	{attribute 'TcIecLibraryType'}
	{attribute 'external_name' := 'F_VN_CalibrateLinescanCameraExp_GUID_4214EBFD_93AA_4917_F265_40A1261014F9'}
	(* Compute the camera parameters (intrinsic + extrinsic) by evaluating images containing a line calibration pattern. The pattern must consist of alternating vertical and diagonal lines, with each diagonal having the same constant slope: |\|\|...\|. The results are only valid for the x-direction of a line scan image. To get accurate x-values for a transformation into world coordinates, the y-coordinate must be set to half the sensor width and so equal to the cy-value of the camera matrix. For other y-values, the results are approximated and can be inaccurate. The extrinsic parameters are computed for the first image in the array. (expert function) *)
	FUNCTION F_VN_CalibrateLinescanCameraExp : HRESULT
	VAR_INPUT
		pSrcImages	:	PVOID;	(* Pointer to an array of 1 or more source images (1 channel). If the images have more than 1 row, each row must contain an image of the same pattern position. *)
		nSrcArraySize	:	UINT;	(* pSrcImages array size *)
		ipPatternLineOrigins	:	ITcVnContainer;	(* X position of the pattern line origins (ContainerType_Vector_REAL, usually same origin for vertical and following diagonal line) *)
		fSlopeRad	:	LREAL;	(* Slope of the diagonal line in rad (> 0, < PI/2), relative to the vertical line (i.e., 0 would be a vertical line, PI/2 a horizontal line) *)
	END_VAR
	VAR_IN_OUT
		aCameraMatrix	:	TcVnMatrix3x3_LREAL;	(* Returns the camera matrix *)
		aDistortionCoefficients	:	TcVnArray8_LREAL;	(* Returns the lens distortion coefficients [k1, k2, p1, p2, k3, k4, k5, k6] *)
		aRotationMatrix	:	TcVnMatrix3x3_LREAL;	(* Returns the rotation matrix *)
		aTranslationVector	:	TcVnVector3_LREAL;	(* Returns the translation vector *)
		fReprojError	:	LREAL;	(* Returns the reprojection error *)
		stCalibrationOptions	:	TcVnCameraCalibrationOptions;	(* Calibration options (recommended to set bFixAspectRatio, bFixPrincipalPoint, bZeroTangentDist) *)
	END_VAR
	VAR_INPUT
		eEdgeDirection	:	ETcVnEdgeDirection;	(* Specification of the edge direction to search for *)
		fMinStrength	:	REAL;	(* Specification of the minimum strength (intensity difference) of the edge to search for *)
		nMaxSearchLines	:	UDINT;	(* Maximum number of search lines (equally distributed over the image height, at most 1 searchline per image row) *)
		nMaxThickness	:	UDINT;	(* Specification of the maximum thickness of the edge to search for, which means fMinStrength must be reached within nMaxThickness pixels *)
		nSubpixelsIterations	:	UDINT;	(* Specifies the number of subpixels (for INTERPOLATION, 10 - 20 usually is sufficient) or maximum number of iterations for optimizing the parameters (for APPROX_ERF and APPROX_GAUSSIAN, 50 - 100 usually is sufficient) *)
		fApproxPrecision	:	REAL;	(* Specifies the approximation precision for APPROX_ERF and APPROX_GAUSSIAN (0.001 usually is sufficient, unused for INTERPOLATION) *)
		eAlgorithm	:	ETcVnEdgeDetectionAlgorithm;	(* Selection of the edge detection algorithm *)
		hrPrev	:	HRESULT;	(* HRESULT indicating the result of previous operations (If SUCCEEDED(hrPrev) equals false, no operation is executed.) *)
	END_VAR

END_FUNCTION

// Functions/Geometric and Coordinate Transformations/Calibration/F_VN_CompensateLensDistortion

	{attribute 'TcIecLibraryType'}
	{attribute 'external_name' := 'F_VN_CompensateLensDistortion_GUID_A7E90272_F769_427D_ED4C_EA7B5F41935C'}
	(* Transforms an image to compensate the lens distortion. *)
	FUNCTION F_VN_CompensateLensDistortion : HRESULT
	VAR_INPUT
		ipSrcImage	:	ITcVnImage;	(* Source image *)
		ipDestImage	:	REFERENCE TO ITcVnImage;	(* Destination image (An appropriate destination image will be created if required.) *)
	END_VAR
	VAR_IN_OUT
		aCameraMatrix	:	TcVnMatrix3x3_LREAL;	(* Camera matrix containing the intrinsic parameters *)
		aDistortionCoefficients	:	TcVnArray4_LREAL;	(* Lens distortion coefficients [k1, k2, p1, p2] *)
	END_VAR
	VAR_INPUT
		hrPrev	:	HRESULT;	(* HRESULT indicating the result of previous operations (If SUCCEEDED(hrPrev) equals false, no operation is executed.) *)
	END_VAR

END_FUNCTION

// Functions/Geometric and Coordinate Transformations/Calibration/F_VN_CompensateLensDistortionExp1

	{attribute 'TcIecLibraryType'}
	{attribute 'external_name' := 'F_VN_CompensateLensDistortionExp1_GUID_3D946475_AB4A_4E66_EAD8_FDBE1E19AFDC'}
	(* Transforms an image to compensate the lens distortion. (expert function) *)
	FUNCTION F_VN_CompensateLensDistortionExp1 : HRESULT
	VAR_INPUT
		ipSrcImage	:	ITcVnImage;	(* Source image *)
		ipDestImage	:	REFERENCE TO ITcVnImage;	(* Destination image (An appropriate destination image will be created if required.) *)
	END_VAR
	VAR_IN_OUT
		aCameraMatrix	:	TcVnMatrix3x3_LREAL;	(* Camera matrix containing the intrinsic parameters *)
		aDistortionCoefficients	:	TcVnArray8_LREAL;	(* Lens distortion coefficients [k1, k2, p1, p2, k3, k4, k5, k6] *)
	END_VAR
	VAR_INPUT
		hrPrev	:	HRESULT;	(* HRESULT indicating the result of previous operations (If SUCCEEDED(hrPrev) equals false, no operation is executed.) *)
	END_VAR

END_FUNCTION

// Functions/Geometric and Coordinate Transformations/Calibration/F_VN_CompensateLensDistortionExp2

	{attribute 'TcIecLibraryType'}
	{attribute 'external_name' := 'F_VN_CompensateLensDistortionExp2_GUID_C20F3BF9_EE4F_4E64_CEDC_52B963B053AC'}
	(* Transforms an image to compensate the lens distortion. (expert function) *)
	FUNCTION F_VN_CompensateLensDistortionExp2 : HRESULT
	VAR_INPUT
		ipSrcImage	:	ITcVnImage;	(* Source image *)
		ipDestImage	:	REFERENCE TO ITcVnImage;	(* Destination image (An appropriate destination image will be created if required.) *)
	END_VAR
	VAR_IN_OUT
		aCameraMatrix	:	TcVnMatrix3x3_LREAL;	(* Camera matrix containing the intrinsic parameters *)
		aDistortionCoefficients	:	TcVnArray8_LREAL;	(* Lens distortion coefficients [k1, k2, p1, p2, k3, k4, k5, k6] *)
		aNewCameraMatrix	:	TcVnMatrix3x3_LREAL;	(* Allows additional scaling and shifting of the result image *)
	END_VAR
	VAR_INPUT
		hrPrev	:	HRESULT;	(* HRESULT indicating the result of previous operations (If SUCCEEDED(hrPrev) equals false, no operation is executed.) *)
	END_VAR

END_FUNCTION

// Functions/Geometric and Coordinate Transformations/Calibration/F_VN_CompensateLensDistortionForPoints

	{attribute 'TcIecLibraryType'}
	{attribute 'external_name' := 'F_VN_CompensateLensDistortionForPoints_GUID_1A71B91E_10E3_4E50_D6FD_7DACBEC96CC6'}
	(* Transforms point coordinates to compensate the lens distortion. *)
	FUNCTION F_VN_CompensateLensDistortionForPoints : HRESULT
	VAR_INPUT
		ipSrcPoints	:	ITcVnContainer;	(* Container with source point coordinates (ContainerType_Vector_TcVnPoint2_REAL or ContainerType_Vector_TcVnPoint2_DINT) *)
		ipDestPoints	:	REFERENCE TO ITcVnContainer;	(* Returns a container with the transformed point coordinates (ContainerType_Vector_TcVnPoint2_REAL) *)
	END_VAR
	VAR_IN_OUT
		aCameraMatrix	:	TcVnMatrix3x3_LREAL;	(* Camera matrix containing the intrinsic parameters *)
		aDistortionCoefficients	:	TcVnArray4_LREAL;	(* Lens distortion coefficients [k1, k2, p1, p2] *)
	END_VAR
	VAR_INPUT
		hrPrev	:	HRESULT;	(* HRESULT indicating the result of previous operations (If SUCCEEDED(hrPrev) equals false, no operation is executed.) *)
	END_VAR

END_FUNCTION

// Functions/Geometric and Coordinate Transformations/Calibration/F_VN_CompensateLensDistortionForPointsExp1

	{attribute 'TcIecLibraryType'}
	{attribute 'external_name' := 'F_VN_CompensateLensDistortionForPointsExp1_GUID_7B846EAA_13D4_4E78_E7DF_523567D8C748'}
	(* Transforms point coordinates to compensate the lens distortion. (expert function) *)
	FUNCTION F_VN_CompensateLensDistortionForPointsExp1 : HRESULT
	VAR_INPUT
		ipSrcPoints	:	ITcVnContainer;	(* Container with source point coordinates (ContainerType_Vector_TcVnPoint2_REAL or ContainerType_Vector_TcVnPoint2_DINT) *)
		ipDestPoints	:	REFERENCE TO ITcVnContainer;	(* Returns a container with the transformed point coordinates (ContainerType_Vector_TcVnPoint2_REAL) *)
	END_VAR
	VAR_IN_OUT
		aCameraMatrix	:	TcVnMatrix3x3_LREAL;	(* Camera matrix containing the intrinsic parameters *)
		aDistortionCoefficients	:	TcVnArray8_LREAL;	(* Lens distortion coefficients [k1, k2, p1, p2, k3, k4, k5, k6] *)
	END_VAR
	VAR_INPUT
		hrPrev	:	HRESULT;	(* HRESULT indicating the result of previous operations (If SUCCEEDED(hrPrev) equals false, no operation is executed.) *)
	END_VAR

END_FUNCTION

// Functions/Geometric and Coordinate Transformations/Calibration/F_VN_CompensateLensDistortionForPointsExp2

	{attribute 'TcIecLibraryType'}
	{attribute 'external_name' := 'F_VN_CompensateLensDistortionForPointsExp2_GUID_34553A45_A6A3_444C_C55B_DC9387F7369D'}
	(* Transforms point coordinates to compensate the lens distortion. (expert function) *)
	FUNCTION F_VN_CompensateLensDistortionForPointsExp2 : HRESULT
	VAR_INPUT
		ipSrcPoints	:	ITcVnContainer;	(* Container with source point coordinates (ContainerType_Vector_TcVnPoint2_REAL or ContainerType_Vector_TcVnPoint2_DINT) *)
		ipDestPoints	:	REFERENCE TO ITcVnContainer;	(* Returns a container with the transformed point coordinates (ContainerType_Vector_TcVnPoint2_REAL) *)
	END_VAR
	VAR_IN_OUT
		aCameraMatrix	:	TcVnMatrix3x3_LREAL;	(* Camera matrix containing the intrinsic parameters *)
		aDistortionCoefficients	:	TcVnArray8_LREAL;	(* Lens distortion coefficients [k1, k2, p1, p2, k3, k4, k5, k6] *)
		aNewCameraMatrix	:	TcVnMatrix3x3_LREAL;	(* Allows additional shifting of the result point coordinates *)
	END_VAR
	VAR_INPUT
		hrPrev	:	HRESULT;	(* HRESULT indicating the result of previous operations (If SUCCEEDED(hrPrev) equals false, no operation is executed.) *)
	END_VAR

END_FUNCTION

// Functions/Geometric and Coordinate Transformations/Calibration/F_VN_DetectPatternPoints

	{attribute 'TcIecLibraryType'}
	{attribute 'external_name' := 'F_VN_DetectPatternPoints_GUID_E1BA4EA3_C273_48EA_C92C_C13F9E969AAA'}
	(* Detects calibration pattern points (circles) within the provided image. *)
	FUNCTION F_VN_DetectPatternPoints : HRESULT
	VAR_INPUT
		ipSrcImage	:	ITcVnImage;	(* Source image (USINT, 1 channel) *)
		ipPatternPoints	:	REFERENCE TO ITcVnContainer;	(* Returns the pattern point positions (ContainerType_Vector_TcVnPoint2_REAL; Non-zero interface pointers are reused.) *)
	END_VAR
	VAR_IN_OUT
		stBlobDetectionParams	:	TcVnParamsBlobDetection;	(* Parameters to detect and filter contours. *)
	END_VAR
	VAR_INPUT
		nNumberOfPoints	:	UDINT;	(* Expected number of pattern points *)
		hrPrev	:	HRESULT;	(* HRESULT indicating the result of previous operations (If SUCCEEDED(hrPrev) equals false, no operation is executed.) *)
	END_VAR

END_FUNCTION

// Functions/Geometric and Coordinate Transformations/Calibration/F_VN_DetectPatternPointsExp

	{attribute 'TcIecLibraryType'}
	{attribute 'external_name' := 'F_VN_DetectPatternPointsExp_GUID_0FD53513_A53D_46BB_DEE5_D943CEECBF42'}
	(* Detects calibration pattern points (circles) within the provided image. (expert function) *)
	FUNCTION F_VN_DetectPatternPointsExp : HRESULT
	VAR_INPUT
		ipSrcImage	:	ITcVnImage;	(* Source image (USINT, 1 channel) *)
		ipPatternPoints	:	REFERENCE TO ITcVnContainer;	(* Returns the pattern point positions (ContainerType_Vector_TcVnPoint2_REAL; Non-zero interface pointers are reused.) *)
	END_VAR
	VAR_IN_OUT
		stBlobDetectionParams	:	TcVnParamsBlobDetection;	(* Parameters to detect and filter contours. *)
	END_VAR
	VAR_INPUT
		nNumberOfPoints	:	UDINT;	(* Expected number of pattern points *)
		fSizeDiffThresFactor	:	REAL;	(* Threshold for filtering contours by average size *)
		bSubpixelAccuracy	:	BOOL;	(* If true, the pattern points are detected with subpixel accuracy *)
		eEdgeDirection	:	ETcVnEdgeDirection;	(* Specification of the edge direction to search for (from center to outside circle) *)
		fMinStrength	:	REAL;	(* Specification of the minimum strength (intensity difference) of the edge to search for *)
		nMaxThickness	:	UDINT;	(* Specification of the maximum thickness of the edge to search for, which means fMinStrength must be reached within nMaxThickness pixels *)
		nSubpixelsIterations	:	UDINT;	(* Specifies the number of subpixels (for INTERPOLATION, 10 - 20 usually is sufficient) or maximum number of iterations for optimizing the parameters (for APPROX_ERF and APPROX_GAUSSIAN, 50 - 100 usually is sufficient) *)
		nSearchLines	:	UDINT;	(* Specifies the amount of search lines, which are equally distributed in all directions (must be >= 8 and a multiple of 4) *)
		fApproxPrecision	:	REAL;	(* Specifies the approximation precision for APPROX_ERF and APPROX_GAUSSIAN (0.001 usually is sufficient, unused for INTERPOLATION) *)
		eAlgorithm	:	ETcVnEdgeDetectionAlgorithm;	(* Selection of the edge detection algorithm *)
		hrPrev	:	HRESULT;	(* HRESULT indicating the result of previous operations (If SUCCEEDED(hrPrev) equals false, no operation is executed.) *)
	END_VAR

END_FUNCTION

// Functions/Geometric and Coordinate Transformations/Calibration/F_VN_GenerateCalibrationPatternReferencePoints

	{attribute 'TcIecLibraryType'}
	{attribute 'external_name' := 'F_VN_GenerateCalibrationPatternReferencePoints_GUID_599A364B_79C4_437C_C2A7_ACD3D87798EB'}
	(* Generate reference points for common calibration patterns. *)
	FUNCTION F_VN_GenerateCalibrationPatternReferencePoints : HRESULT
	VAR_INPUT
		ipReferencePoints	:	REFERENCE TO ITcVnContainer;	(* Returns the generated reference points (ContainerType_Vector_TcVnPoint3_REAL) *)
		ePattern	:	ETcVnCalibrationPattern;	(* Calibration pattern type *)
		eOrigin	:	ETcVnCalibrationPatternOrigin;	(* Calibration pattern origin *)
		nWidth	:	UDINT;	(* Pattern width, i.e. number of pattern points in x direction *)
		nHeight	:	UDINT;	(* Pattern height, i.e. number of pattern points in y direction *)
		fDistX	:	REAL;	(* Distance between pattern points in x direction *)
		fDistY	:	REAL;	(* Distance between pattern points in y direction *)
		hrPrev	:	HRESULT;	(* HRESULT indicating the result of previous operations (If SUCCEEDED(hrPrev) equals false, no operation is executed.) *)
	END_VAR

END_FUNCTION

// Functions/Geometric and Coordinate Transformations/Calibration/F_VN_ImagePointsWorldDistance

	{attribute 'TcIecLibraryType'}
	{attribute 'external_name' := 'F_VN_ImagePointsWorldDistance_GUID_07588962_595D_4F8E_F6BA_08B6D70B97B0'}
	(* Computes the distance in the world coordinate system between two points (in the same world coordinate z layer) given in image coordinates. *)
	FUNCTION F_VN_ImagePointsWorldDistance : HRESULT
	VAR_IN_OUT
		aImagePoint1	:	TcVnPoint2_REAL;	(* First point in the image coordinate system *)
		aImagePoint2	:	TcVnPoint2_REAL;	(* Second point in the image coordinate system *)
		fWorldDistance	:	LREAL;	(* Returns the distance between aImagePoint1 and aImagePoint2 in the world coordinate system *)
		aCameraMatrix	:	TcVnMatrix3x3_LREAL;	(* 3x3 camera matrix containing the intrinsic parameters *)
		aDistortionCoefficients	:	TcVnArray8_LREAL;	(* Lens distortion coefficients [k1, k2, p1, p2, k3, k4, k5, k6] *)
		aRotationMatrix	:	TcVnMatrix3x3_LREAL;	(* 3x3 rotation matrix *)
		aTranslationVector	:	TcVnVector3_LREAL;	(* Translation vector *)
	END_VAR
	VAR_INPUT
		fZ	:	LREAL;	(* z coordinate (world coordinate system) of the given points (0 would be at (toplevel) calibration pattern) *)
		hrPrev	:	HRESULT;	(* HRESULT indicating the result of previous operations (If SUCCEEDED(hrPrev) equals false, no operation is executed.) *)
	END_VAR

END_FUNCTION

// Functions/Geometric and Coordinate Transformations/Calibration/F_VN_SolvePnP

	{attribute 'TcIecLibraryType'}
	{attribute 'external_name' := 'F_VN_SolvePnP_GUID_4CDE4046_D05B_41CC_F0BB_C7149D9A0102'}
	(* Computes the rotation matrix and translation vector from 3D-2D point correspondences. *)
	FUNCTION F_VN_SolvePnP : HRESULT
	VAR_INPUT
		ipImagePoints	:	ITcVnContainer;	(* Image points (ContainerType_Vector_TcVnPoint2_REAL, requires at least 4 points in the same order as in ipReferencePoints) *)
		ipReferencePoints	:	ITcVnContainer;	(* Reference world points (ContainerType_Vector_TcVnPoint3_REAL, same number of points as in ipImagePoints) *)
	END_VAR
	VAR_IN_OUT
		aCameraMatrix	:	TcVnMatrix3x3_LREAL;	(* Camera matrix (e.g. computed with one of the CalibrateCamera functions) *)
		aDistortionCoefficients	:	TcVnArray8_LREAL;	(* Lens distortion coefficients [k1, k2, p1, p2, k3, k4, k5, k6] (e.g. computed with one of the CalibrateCamera functions) *)
		aRotationMatrix	:	TcVnMatrix3x3_LREAL;	(* Returns the rotation matrix *)
		aTranslationVector	:	TcVnVector3_LREAL;	(* Returns the translation vector *)
		fReprojError	:	LREAL;	(* Returns the reprojection error *)
	END_VAR
	VAR_INPUT
		hrPrev	:	HRESULT;	(* HRESULT indicating the result of previous operations (If SUCCEEDED(hrPrev) equals false, no operation is executed.) *)
	END_VAR

END_FUNCTION

// Functions/Geometric and Coordinate Transformations/Calibration/F_VN_SolvePnPExp

	{attribute 'TcIecLibraryType'}
	{attribute 'external_name' := 'F_VN_SolvePnPExp_GUID_4E0700BF_599A_43BB_DEA5_C384C8638085'}
	(* Computes the rotation matrix and translation vector from 3D-2D point correspondences. (expert function) *)
	FUNCTION F_VN_SolvePnPExp : HRESULT
	VAR_INPUT
		ipImagePoints	:	ITcVnContainer;	(* Image points (ContainerType_Vector_TcVnPoint2_REAL, requires at least 4 points in the same order as in ipReferencePoints) *)
		ipReferencePoints	:	ITcVnContainer;	(* Reference world points (ContainerType_Vector_TcVnPoint3_REAL, same number of points as in ipImagePoints) *)
	END_VAR
	VAR_IN_OUT
		aCameraMatrix	:	TcVnMatrix3x3_LREAL;	(* Camera matrix (e.g. computed with one of the CalibrateCamera functions) *)
		aDistortionCoefficients	:	TcVnArray8_LREAL;	(* Lens distortion coefficients [k1, k2, p1, p2, k3, k4, k5, k6] (e.g. computed with one of the CalibrateCamera functions) *)
		aRotationMatrix	:	TcVnMatrix3x3_LREAL;	(* Returns the rotation matrix *)
		aTranslationVector	:	TcVnVector3_LREAL;	(* Returns the translation vector *)
		fReprojError	:	LREAL;	(* Returns the reprojection error *)
	END_VAR
	VAR_INPUT
		eMethod	:	ETcVnSolvePnPMethod;	(* Solve PnP method *)
		bUseExtrinsicGuess	:	BOOL;	(* If true, the provided rotation matrix and translation vector are used as an initial guess for further optimization (only supported for the SPM_ITERATIVE method). *)
		hrPrev	:	HRESULT;	(* HRESULT indicating the result of previous operations (If SUCCEEDED(hrPrev) equals false, no operation is executed.) *)
	END_VAR

END_FUNCTION

// Functions/Geometric and Coordinate Transformations/Calibration/F_VN_SortDetectedPatternPoints

	{attribute 'TcIecLibraryType'}
	{attribute 'external_name' := 'F_VN_SortDetectedPatternPoints_GUID_A5133D21_0CC3_4002_DB54_EEBCCDC9DF91'}
	(* Sort the detected pattern points according to the relative positions of the calibration pattern points. *)
	FUNCTION F_VN_SortDetectedPatternPoints : HRESULT
	VAR_INPUT
		ipImagePoints	:	ITcVnContainer;	(* Detected pattern point positions in the image coordinate system (will be sorted by this function, ContainerType_Vector_TcVnPoint2_REAL) *)
		ipPatternPoints	:	ITcVnContainer;	(* The pattern points in the calibration pattern coordinate system, used as a reference to sort ipImagePoints (ContainerType_Vector_TcVnPoint3_REAL) *)
		hrPrev	:	HRESULT;	(* HRESULT indicating the result of previous operations (If SUCCEEDED(hrPrev) equals false, no operation is executed.) *)
	END_VAR

END_FUNCTION

// Functions/Geometric and Coordinate Transformations/Calibration/F_VN_TransformCoordinatesPlanar_Container

	{attribute 'TcIecLibraryType'}
	{attribute 'external_name' := 'F_VN_TransformCoordinatesPlanar_Container_GUID_67542BE0_71A3_4501_F6F6_3E1455460A09'}
	(* Compute real-world coordinates for given image points or vice versa. *)
	FUNCTION F_VN_TransformCoordinatesPlanar_Container : HRESULT
	VAR_INPUT
		ipSrcPoints	:	ITcVnContainer;	(* Container with 2D source points (TcVnPoint2_DINT or TcVnPoint2_REAL or TcVnPoint2_LREAL) *)
		ipDestPoints	:	REFERENCE TO ITcVnContainer;	(* Returns the transformed 2D points (TcVnPoint2_LREAL) *)
	END_VAR
	VAR_IN_OUT
		aTransformationMatrix	:	TcVnMatrix3x3_LREAL;	(* Transformation matrix obtained with VnCalibrateCameraPlanar() or its inverse matrix obtained with VnInvertMatrix3x3() *)
	END_VAR
	VAR_INPUT
		hrPrev	:	HRESULT;	(* HRESULT indicating the result of previous operations (If SUCCEEDED(hrPrev) equals false, no operation is executed.) *)
	END_VAR

END_FUNCTION

// Functions/Geometric and Coordinate Transformations/Calibration/F_VN_TransformCoordinatesPlanar_Point

	{attribute 'TcIecLibraryType'}
	{attribute 'external_name' := 'F_VN_TransformCoordinatesPlanar_Point_GUID_93AE96FC_5E50_46EB_F82A_EF8661198BF3'}
	(* Compute real-world coordinates for a given image point or vice versa. *)
	FUNCTION F_VN_TransformCoordinatesPlanar_Point : HRESULT
	VAR_IN_OUT
		aSrcPoint	:	TcVnPoint2_LREAL;	(* Point in the source coordinate system *)
		aDestPoint	:	TcVnPoint2_LREAL;	(* Returns point in the destination coordinate system *)
		aTransformationMatrix	:	TcVnMatrix3x3_LREAL;	(* Transformation matrix obtained with VnCalibrateCameraPlanar() or its inverse matrix obtained with VnInvertMatrix3x3() *)
	END_VAR
	VAR_INPUT
		hrPrev	:	HRESULT;	(* HRESULT indicating the result of previous operations (If SUCCEEDED(hrPrev) equals false, no operation is executed.) *)
	END_VAR

END_FUNCTION

// Functions/Geometric and Coordinate Transformations/Calibration/F_VN_TransformCoordinatesImageToWorld_Container

	{attribute 'TcIecLibraryType'}
	{attribute 'external_name' := 'F_VN_TransformCoordinatesImageToWorld_Container_GUID_54C38E15_05D5_44A4_C9DC_F641ACBFF843'}
	(* Transform 2D image point coordinates to 3D world coordinates (using intrinsic + extrinsic calibration results). *)
	FUNCTION F_VN_TransformCoordinatesImageToWorld_Container : HRESULT
	VAR_INPUT
		ipSrcPoints2D	:	ITcVnContainer;	(* Container with 2D source points (TcVnPoint2_DINT or TcVnPoint2_REAL or TcVnPoint2_LREAL) *)
		ipDestPoints3D	:	REFERENCE TO ITcVnContainer;	(* Returns the transformed 3D points (TcVnPoint3_LREAL) *)
	END_VAR
	VAR_IN_OUT
		aCameraMatrix	:	TcVnMatrix3x3_LREAL;	(* 3x3 camera matrix containing the intrinsic parameters *)
		aDistortionCoefficients	:	TcVnArray8_LREAL;	(* Lens distortion coefficients [k1, k2, p1, p2, k3, k4, k5, k6] *)
		aRotationMatrix	:	TcVnMatrix3x3_LREAL;	(* 3x3 rotation matrix *)
		aTranslationVector	:	TcVnVector3_LREAL;	(* Translation vector *)
	END_VAR
	VAR_INPUT
		fZ	:	LREAL;	(* z coordinate (world coordinate system) of the transformed points (0 would be at (toplevel) calibration pattern) *)
		hrPrev	:	HRESULT;	(* HRESULT indicating the result of previous operations (If SUCCEEDED(hrPrev) equals false, no operation is executed.) *)
	END_VAR

END_FUNCTION

// Functions/Geometric and Coordinate Transformations/Calibration/F_VN_TransformCoordinatesImageToWorld_Point

	{attribute 'TcIecLibraryType'}
	{attribute 'external_name' := 'F_VN_TransformCoordinatesImageToWorld_Point_GUID_83E167E3_3126_4560_FF31_E7D52361951D'}
	(* Transform 2D image point coordinate to 3D world coordinate (using intrinsic + extrinsic calibration results). *)
	FUNCTION F_VN_TransformCoordinatesImageToWorld_Point : HRESULT
	VAR_IN_OUT
		aSrcPoint	:	TcVnPoint2_LREAL;	(* Point in the image coordinate system *)
		aDestPoint	:	TcVnPoint3_LREAL;	(* Returns the point in the world coordinate system *)
		aCameraMatrix	:	TcVnMatrix3x3_LREAL;	(* 3x3 camera matrix containing the intrinsic parameters *)
		aDistortionCoefficients	:	TcVnArray8_LREAL;	(* Lens distortion coefficients [k1, k2, p1, p2, k3, k4, k5, k6] *)
		aRotationMatrix	:	TcVnMatrix3x3_LREAL;	(* 3x3 rotation matrix *)
		aTranslationVector	:	TcVnVector3_LREAL;	(* Translation vector *)
	END_VAR
	VAR_INPUT
		fZ	:	LREAL;	(* z coordinate (world coordinate system) of the transformed points (0 would be at (toplevel) calibration pattern) *)
		hrPrev	:	HRESULT;	(* HRESULT indicating the result of previous operations (If SUCCEEDED(hrPrev) equals false, no operation is executed.) *)
	END_VAR

END_FUNCTION

// Functions/Geometric and Coordinate Transformations/Calibration/F_VN_TransformCoordinatesWorldToImage_Container

	{attribute 'TcIecLibraryType'}
	{attribute 'external_name' := 'F_VN_TransformCoordinatesWorldToImage_Container_GUID_C6D59311_1ED5_4B28_FFA0_497C13CE1463'}
	(* Transform 3D world coordinates to 2D image coordinates (using intrinsic + extrinsic calibration results). *)
	FUNCTION F_VN_TransformCoordinatesWorldToImage_Container : HRESULT
	VAR_INPUT
		ipSrcPoints3D	:	ITcVnContainer;	(* Container with 3D source points (TcVnPoint3_LREAL) *)
		ipDestPoints2D	:	REFERENCE TO ITcVnContainer;	(* Returns the transformed 2D points (TcVnPoint2_REAL or TcVnPoint2_DINT, depending on bInteger) *)
	END_VAR
	VAR_IN_OUT
		aCameraMatrix	:	TcVnMatrix3x3_LREAL;	(* 3x3 camera matrix containing the intrinsic parameters *)
		aDistortionCoefficients	:	TcVnArray8_LREAL;	(* Lens distortion coefficients [k1, k2, p1, p2, k3, k4, k5, k6] *)
		aRotationMatrix	:	TcVnMatrix3x3_LREAL;	(* 3x3 rotation matrix *)
		aTranslationVector	:	TcVnVector3_LREAL;	(* Translation vector *)
	END_VAR
	VAR_INPUT
		bInteger	:	BOOL;	(* Selects whether the function returns a container of TcVnPoint2_DINT or TcVnPoint2_REAL *)
		hrPrev	:	HRESULT;	(* HRESULT indicating the result of previous operations (If SUCCEEDED(hrPrev) equals false, no operation is executed.) *)
	END_VAR

END_FUNCTION

// Functions/Geometric and Coordinate Transformations/Calibration/F_VN_TransformCoordinatesWorldToImage_Point

	{attribute 'TcIecLibraryType'}
	{attribute 'external_name' := 'F_VN_TransformCoordinatesWorldToImage_Point_GUID_82E7FA31_3D31_404A_FDFF_B82253ED906D'}
	(* Transform 3D world coordinates to 2D image coordinates (using intrinsic + extrinsic calibration results). *)
	FUNCTION F_VN_TransformCoordinatesWorldToImage_Point : HRESULT
	VAR_IN_OUT
		aSrcPoint	:	TcVnPoint3_LREAL;	(* 3D source point (world coordinate system) *)
		aDestPoint	:	TcVnPoint2_REAL;	(* Returns the transformed 2D point (image coordinate system) *)
		aCameraMatrix	:	TcVnMatrix3x3_LREAL;	(* 3x3 camera matrix containing the intrinsic parameters *)
		aDistortionCoefficients	:	TcVnArray8_LREAL;	(* Lens distortion coefficients [k1, k2, p1, p2, k3, k4, k5, k6] *)
		aRotationMatrix	:	TcVnMatrix3x3_LREAL;	(* 3x3 rotation matrix *)
		aTranslationVector	:	TcVnVector3_LREAL;	(* Translation vector *)
	END_VAR
	VAR_INPUT
		hrPrev	:	HRESULT;	(* HRESULT indicating the result of previous operations (If SUCCEEDED(hrPrev) equals false, no operation is executed.) *)
	END_VAR

END_FUNCTION

// Functions/Container Statistics/F_VN_MaxElementElementwise/F_VN_MaxElementElementwise_DINT

	{attribute 'TcIecLibraryType'}
	{attribute 'external_name' := 'F_VN_MaxElementElementwise_DINT_GUID_A5D21510_D344_4EA5_C76D_A584DA80E7CB'}
	(* Gets the element wise maximum container element. *)
	FUNCTION F_VN_MaxElementElementwise_DINT : HRESULT
	VAR_INPUT
		ipContainer	:	ITcVnContainer;	(* Source container *)
	END_VAR
	VAR_IN_OUT
		nMax	:	DINT;	(* Returns the requested element *)
	END_VAR
	VAR_INPUT
		hrPrev	:	HRESULT;	(* HRESULT indicating the result of previous operations (If SUCCEEDED(hrPrev) equals false, no operation is executed.) *)
	END_VAR

END_FUNCTION

// Functions/Container Statistics/F_VN_MaxElementElementwise/F_VN_MaxElementElementwise_INT

	{attribute 'TcIecLibraryType'}
	{attribute 'external_name' := 'F_VN_MaxElementElementwise_INT_GUID_91DB98A7_6687_4D0E_FC88_E57CE322951B'}
	(* Gets the element wise maximum container element. *)
	FUNCTION F_VN_MaxElementElementwise_INT : HRESULT
	VAR_INPUT
		ipContainer	:	ITcVnContainer;	(* Source container *)
	END_VAR
	VAR_IN_OUT
		nMax	:	INT;	(* Returns the requested element *)
	END_VAR
	VAR_INPUT
		hrPrev	:	HRESULT;	(* HRESULT indicating the result of previous operations (If SUCCEEDED(hrPrev) equals false, no operation is executed.) *)
	END_VAR

END_FUNCTION

// Functions/Container Statistics/F_VN_MaxElementElementwise/F_VN_MaxElementElementwise_LREAL

	{attribute 'TcIecLibraryType'}
	{attribute 'external_name' := 'F_VN_MaxElementElementwise_LREAL_GUID_46666C73_74A0_41C9_FD1B_24334D2A3765'}
	(* Gets the element wise maximum container element. *)
	FUNCTION F_VN_MaxElementElementwise_LREAL : HRESULT
	VAR_INPUT
		ipContainer	:	ITcVnContainer;	(* Source container *)
	END_VAR
	VAR_IN_OUT
		fMax	:	LREAL;	(* Returns the requested element *)
	END_VAR
	VAR_INPUT
		hrPrev	:	HRESULT;	(* HRESULT indicating the result of previous operations (If SUCCEEDED(hrPrev) equals false, no operation is executed.) *)
	END_VAR

END_FUNCTION

// Functions/Container Statistics/F_VN_MaxElementElementwise/F_VN_MaxElementElementwise_REAL

	{attribute 'TcIecLibraryType'}
	{attribute 'external_name' := 'F_VN_MaxElementElementwise_REAL_GUID_2D97D886_E0C1_4CEA_F01B_CF80CC07EDEB'}
	(* Gets the element wise maximum container element. *)
	FUNCTION F_VN_MaxElementElementwise_REAL : HRESULT
	VAR_INPUT
		ipContainer	:	ITcVnContainer;	(* Source container *)
	END_VAR
	VAR_IN_OUT
		fMax	:	REAL;	(* Returns the requested element *)
	END_VAR
	VAR_INPUT
		hrPrev	:	HRESULT;	(* HRESULT indicating the result of previous operations (If SUCCEEDED(hrPrev) equals false, no operation is executed.) *)
	END_VAR

END_FUNCTION

// Functions/Container Statistics/F_VN_MaxElementElementwise/F_VN_MaxElementElementwise_SINT

	{attribute 'TcIecLibraryType'}
	{attribute 'external_name' := 'F_VN_MaxElementElementwise_SINT_GUID_D306F3D3_3CF3_43E6_D738_820C4BAADC11'}
	(* Gets the element wise maximum container element. *)
	FUNCTION F_VN_MaxElementElementwise_SINT : HRESULT
	VAR_INPUT
		ipContainer	:	ITcVnContainer;	(* Source container *)
	END_VAR
	VAR_IN_OUT
		nMax	:	SINT;	(* Returns the requested element *)
	END_VAR
	VAR_INPUT
		hrPrev	:	HRESULT;	(* HRESULT indicating the result of previous operations (If SUCCEEDED(hrPrev) equals false, no operation is executed.) *)
	END_VAR

END_FUNCTION

// Functions/Container Statistics/F_VN_MaxElementElementwise/F_VN_MaxElementElementwise_TcVnPoint2_DINT

	{attribute 'TcIecLibraryType'}
	{attribute 'external_name' := 'F_VN_MaxElementElementwise_TcVnPoint2_DINT_GUID_AFE11F89_F703_4FE4_E53E_6DAE81C1EAC8'}
	(* Gets the element wise maximum container element. *)
	FUNCTION F_VN_MaxElementElementwise_TcVnPoint2_DINT : HRESULT
	VAR_INPUT
		ipContainer	:	ITcVnContainer;	(* Source container *)
	END_VAR
	VAR_IN_OUT
		aMax	:	TcVnPoint2_DINT;	(* Returns the requested element *)
	END_VAR
	VAR_INPUT
		hrPrev	:	HRESULT;	(* HRESULT indicating the result of previous operations (If SUCCEEDED(hrPrev) equals false, no operation is executed.) *)
	END_VAR

END_FUNCTION

// Functions/Container Statistics/F_VN_MaxElementElementwise/F_VN_MaxElementElementwise_TcVnPoint2_LREAL

	{attribute 'TcIecLibraryType'}
	{attribute 'external_name' := 'F_VN_MaxElementElementwise_TcVnPoint2_LREAL_GUID_A18152A5_BBC0_4F75_C048_CB1A64DF6F78'}
	(* Gets the element wise maximum container element. *)
	FUNCTION F_VN_MaxElementElementwise_TcVnPoint2_LREAL : HRESULT
	VAR_INPUT
		ipContainer	:	ITcVnContainer;	(* Source container *)
	END_VAR
	VAR_IN_OUT
		aMax	:	TcVnPoint2_LREAL;	(* Returns the requested element *)
	END_VAR
	VAR_INPUT
		hrPrev	:	HRESULT;	(* HRESULT indicating the result of previous operations (If SUCCEEDED(hrPrev) equals false, no operation is executed.) *)
	END_VAR

END_FUNCTION

// Functions/Container Statistics/F_VN_MaxElementElementwise/F_VN_MaxElementElementwise_TcVnPoint2_REAL

	{attribute 'TcIecLibraryType'}
	{attribute 'external_name' := 'F_VN_MaxElementElementwise_TcVnPoint2_REAL_GUID_0A7850A3_6CBE_4C11_E2C2_A8C8F94223EC'}
	(* Gets the element wise maximum container element. *)
	FUNCTION F_VN_MaxElementElementwise_TcVnPoint2_REAL : HRESULT
	VAR_INPUT
		ipContainer	:	ITcVnContainer;	(* Source container *)
	END_VAR
	VAR_IN_OUT
		aMax	:	TcVnPoint2_REAL;	(* Returns the requested element *)
	END_VAR
	VAR_INPUT
		hrPrev	:	HRESULT;	(* HRESULT indicating the result of previous operations (If SUCCEEDED(hrPrev) equals false, no operation is executed.) *)
	END_VAR

END_FUNCTION

// Functions/Container Statistics/F_VN_MaxElementElementwise/F_VN_MaxElementElementwise_TcVnPoint3_LREAL

	{attribute 'TcIecLibraryType'}
	{attribute 'external_name' := 'F_VN_MaxElementElementwise_TcVnPoint3_LREAL_GUID_0E2D357B_DA71_420C_C182_5BB598D9854A'}
	(* Gets the element wise maximum container element. *)
	FUNCTION F_VN_MaxElementElementwise_TcVnPoint3_LREAL : HRESULT
	VAR_INPUT
		ipContainer	:	ITcVnContainer;	(* Source container *)
	END_VAR
	VAR_IN_OUT
		aMax	:	TcVnPoint3_LREAL;	(* Returns the requested element *)
	END_VAR
	VAR_INPUT
		hrPrev	:	HRESULT;	(* HRESULT indicating the result of previous operations (If SUCCEEDED(hrPrev) equals false, no operation is executed.) *)
	END_VAR

END_FUNCTION

// Functions/Container Statistics/F_VN_MaxElementElementwise/F_VN_MaxElementElementwise_TcVnPoint3_REAL

	{attribute 'TcIecLibraryType'}
	{attribute 'external_name' := 'F_VN_MaxElementElementwise_TcVnPoint3_REAL_GUID_F9F02289_4D77_43A0_C6A9_7BCB711D1487'}
	(* Gets the element wise maximum container element. *)
	FUNCTION F_VN_MaxElementElementwise_TcVnPoint3_REAL : HRESULT
	VAR_INPUT
		ipContainer	:	ITcVnContainer;	(* Source container *)
	END_VAR
	VAR_IN_OUT
		aMax	:	TcVnPoint3_REAL;	(* Returns the requested element *)
	END_VAR
	VAR_INPUT
		hrPrev	:	HRESULT;	(* HRESULT indicating the result of previous operations (If SUCCEEDED(hrPrev) equals false, no operation is executed.) *)
	END_VAR

END_FUNCTION

// Functions/Container Statistics/F_VN_MaxElementElementwise/F_VN_MaxElementElementwise_TcVnVector2_DINT

	{attribute 'TcIecLibraryType'}
	{attribute 'external_name' := 'F_VN_MaxElementElementwise_TcVnVector2_DINT_GUID_C78EA9B8_202F_45EB_D61E_82AFEF30FB02'}
	(* Gets the element wise maximum container element. *)
	FUNCTION F_VN_MaxElementElementwise_TcVnVector2_DINT : HRESULT
	VAR_INPUT
		ipContainer	:	ITcVnContainer;	(* Source container *)
	END_VAR
	VAR_IN_OUT
		aMax	:	TcVnVector2_DINT;	(* Returns the requested element *)
	END_VAR
	VAR_INPUT
		hrPrev	:	HRESULT;	(* HRESULT indicating the result of previous operations (If SUCCEEDED(hrPrev) equals false, no operation is executed.) *)
	END_VAR

END_FUNCTION

// Functions/Container Statistics/F_VN_MaxElementElementwise/F_VN_MaxElementElementwise_TcVnVector2_INT

	{attribute 'TcIecLibraryType'}
	{attribute 'external_name' := 'F_VN_MaxElementElementwise_TcVnVector2_INT_GUID_CE01E54C_7609_4F66_CA92_03A574574092'}
	(* Gets the element wise maximum container element. *)
	FUNCTION F_VN_MaxElementElementwise_TcVnVector2_INT : HRESULT
	VAR_INPUT
		ipContainer	:	ITcVnContainer;	(* Source container *)
	END_VAR
	VAR_IN_OUT
		aMax	:	TcVnVector2_INT;	(* Returns the requested element *)
	END_VAR
	VAR_INPUT
		hrPrev	:	HRESULT;	(* HRESULT indicating the result of previous operations (If SUCCEEDED(hrPrev) equals false, no operation is executed.) *)
	END_VAR

END_FUNCTION

// Functions/Container Statistics/F_VN_MaxElementElementwise/F_VN_MaxElementElementwise_TcVnVector2_REAL

	{attribute 'TcIecLibraryType'}
	{attribute 'external_name' := 'F_VN_MaxElementElementwise_TcVnVector2_REAL_GUID_A91286AE_C599_492D_D68F_DBABD12D5EF9'}
	(* Gets the element wise maximum container element. *)
	FUNCTION F_VN_MaxElementElementwise_TcVnVector2_REAL : HRESULT
	VAR_INPUT
		ipContainer	:	ITcVnContainer;	(* Source container *)
	END_VAR
	VAR_IN_OUT
		aMax	:	TcVnVector2_REAL;	(* Returns the requested element *)
	END_VAR
	VAR_INPUT
		hrPrev	:	HRESULT;	(* HRESULT indicating the result of previous operations (If SUCCEEDED(hrPrev) equals false, no operation is executed.) *)
	END_VAR

END_FUNCTION

// Functions/Container Statistics/F_VN_MaxElementElementwise/F_VN_MaxElementElementwise_TcVnVector2_SINT

	{attribute 'TcIecLibraryType'}
	{attribute 'external_name' := 'F_VN_MaxElementElementwise_TcVnVector2_SINT_GUID_2DCF38B4_B309_4447_F0CB_E7B65E5F123A'}
	(* Gets the element wise maximum container element. *)
	FUNCTION F_VN_MaxElementElementwise_TcVnVector2_SINT : HRESULT
	VAR_INPUT
		ipContainer	:	ITcVnContainer;	(* Source container *)
	END_VAR
	VAR_IN_OUT
		aMax	:	TcVnVector2_SINT;	(* Returns the requested element *)
	END_VAR
	VAR_INPUT
		hrPrev	:	HRESULT;	(* HRESULT indicating the result of previous operations (If SUCCEEDED(hrPrev) equals false, no operation is executed.) *)
	END_VAR

END_FUNCTION

// Functions/Container Statistics/F_VN_MaxElementElementwise/F_VN_MaxElementElementwise_TcVnVector2_UINT

	{attribute 'TcIecLibraryType'}
	{attribute 'external_name' := 'F_VN_MaxElementElementwise_TcVnVector2_UINT_GUID_BF12DB7A_1E3B_4E69_F13F_F1EF18A3023E'}
	(* Gets the element wise maximum container element. *)
	FUNCTION F_VN_MaxElementElementwise_TcVnVector2_UINT : HRESULT
	VAR_INPUT
		ipContainer	:	ITcVnContainer;	(* Source container *)
	END_VAR
	VAR_IN_OUT
		aMax	:	TcVnVector2_UINT;	(* Returns the requested element *)
	END_VAR
	VAR_INPUT
		hrPrev	:	HRESULT;	(* HRESULT indicating the result of previous operations (If SUCCEEDED(hrPrev) equals false, no operation is executed.) *)
	END_VAR

END_FUNCTION

// Functions/Container Statistics/F_VN_MaxElementElementwise/F_VN_MaxElementElementwise_TcVnVector2_USINT

	{attribute 'TcIecLibraryType'}
	{attribute 'external_name' := 'F_VN_MaxElementElementwise_TcVnVector2_USINT_GUID_EA7A133B_9400_484E_F009_6D9FDFE81353'}
	(* Gets the element wise maximum container element. *)
	FUNCTION F_VN_MaxElementElementwise_TcVnVector2_USINT : HRESULT
	VAR_INPUT
		ipContainer	:	ITcVnContainer;	(* Source container *)
	END_VAR
	VAR_IN_OUT
		aMax	:	TcVnVector2_USINT;	(* Returns the requested element *)
	END_VAR
	VAR_INPUT
		hrPrev	:	HRESULT;	(* HRESULT indicating the result of previous operations (If SUCCEEDED(hrPrev) equals false, no operation is executed.) *)
	END_VAR

END_FUNCTION

// Functions/Container Statistics/F_VN_MaxElementElementwise/F_VN_MaxElementElementwise_TcVnVector3_INT

	{attribute 'TcIecLibraryType'}
	{attribute 'external_name' := 'F_VN_MaxElementElementwise_TcVnVector3_INT_GUID_1DECA8A5_47F0_4445_EE05_71916D69E935'}
	(* Gets the element wise maximum container element. *)
	FUNCTION F_VN_MaxElementElementwise_TcVnVector3_INT : HRESULT
	VAR_INPUT
		ipContainer	:	ITcVnContainer;	(* Source container *)
	END_VAR
	VAR_IN_OUT
		aMax	:	TcVnVector3_INT;	(* Returns the requested element *)
	END_VAR
	VAR_INPUT
		hrPrev	:	HRESULT;	(* HRESULT indicating the result of previous operations (If SUCCEEDED(hrPrev) equals false, no operation is executed.) *)
	END_VAR

END_FUNCTION

// Functions/Container Statistics/F_VN_MaxElementElementwise/F_VN_MaxElementElementwise_TcVnVector3_REAL

	{attribute 'TcIecLibraryType'}
	{attribute 'external_name' := 'F_VN_MaxElementElementwise_TcVnVector3_REAL_GUID_9E5A5244_E5A7_4849_E561_A3EDEAE61369'}
	(* Gets the element wise maximum container element. *)
	FUNCTION F_VN_MaxElementElementwise_TcVnVector3_REAL : HRESULT
	VAR_INPUT
		ipContainer	:	ITcVnContainer;	(* Source container *)
	END_VAR
	VAR_IN_OUT
		aMax	:	TcVnVector3_REAL;	(* Returns the requested element *)
	END_VAR
	VAR_INPUT
		hrPrev	:	HRESULT;	(* HRESULT indicating the result of previous operations (If SUCCEEDED(hrPrev) equals false, no operation is executed.) *)
	END_VAR

END_FUNCTION

// Functions/Container Statistics/F_VN_MaxElementElementwise/F_VN_MaxElementElementwise_TcVnVector3_SINT

	{attribute 'TcIecLibraryType'}
	{attribute 'external_name' := 'F_VN_MaxElementElementwise_TcVnVector3_SINT_GUID_FD11B09B_F658_4940_F166_B6D49AC1AA2F'}
	(* Gets the element wise maximum container element. *)
	FUNCTION F_VN_MaxElementElementwise_TcVnVector3_SINT : HRESULT
	VAR_INPUT
		ipContainer	:	ITcVnContainer;	(* Source container *)
	END_VAR
	VAR_IN_OUT
		aMax	:	TcVnVector3_SINT;	(* Returns the requested element *)
	END_VAR
	VAR_INPUT
		hrPrev	:	HRESULT;	(* HRESULT indicating the result of previous operations (If SUCCEEDED(hrPrev) equals false, no operation is executed.) *)
	END_VAR

END_FUNCTION

// Functions/Container Statistics/F_VN_MaxElementElementwise/F_VN_MaxElementElementwise_TcVnVector3_UINT

	{attribute 'TcIecLibraryType'}
	{attribute 'external_name' := 'F_VN_MaxElementElementwise_TcVnVector3_UINT_GUID_88272368_EF0D_447A_DE8F_0748AEB81653'}
	(* Gets the element wise maximum container element. *)
	FUNCTION F_VN_MaxElementElementwise_TcVnVector3_UINT : HRESULT
	VAR_INPUT
		ipContainer	:	ITcVnContainer;	(* Source container *)
	END_VAR
	VAR_IN_OUT
		aMax	:	TcVnVector3_UINT;	(* Returns the requested element *)
	END_VAR
	VAR_INPUT
		hrPrev	:	HRESULT;	(* HRESULT indicating the result of previous operations (If SUCCEEDED(hrPrev) equals false, no operation is executed.) *)
	END_VAR

END_FUNCTION

// Functions/Container Statistics/F_VN_MaxElementElementwise/F_VN_MaxElementElementwise_TcVnVector3_USINT

	{attribute 'TcIecLibraryType'}
	{attribute 'external_name' := 'F_VN_MaxElementElementwise_TcVnVector3_USINT_GUID_55A7DF92_8318_4AF1_EDE1_5673AB931B04'}
	(* Gets the element wise maximum container element. *)
	FUNCTION F_VN_MaxElementElementwise_TcVnVector3_USINT : HRESULT
	VAR_INPUT
		ipContainer	:	ITcVnContainer;	(* Source container *)
	END_VAR
	VAR_IN_OUT
		aMax	:	TcVnVector3_USINT;	(* Returns the requested element *)
	END_VAR
	VAR_INPUT
		hrPrev	:	HRESULT;	(* HRESULT indicating the result of previous operations (If SUCCEEDED(hrPrev) equals false, no operation is executed.) *)
	END_VAR

END_FUNCTION

// Functions/Container Statistics/F_VN_MaxElementElementwise/F_VN_MaxElementElementwise_TcVnVector4_DINT

	{attribute 'TcIecLibraryType'}
	{attribute 'external_name' := 'F_VN_MaxElementElementwise_TcVnVector4_DINT_GUID_52DF9DB5_6BEB_4191_CB71_0352BB8A5426'}
	(* Gets the element wise maximum container element. *)
	FUNCTION F_VN_MaxElementElementwise_TcVnVector4_DINT : HRESULT
	VAR_INPUT
		ipContainer	:	ITcVnContainer;	(* Source container *)
	END_VAR
	VAR_IN_OUT
		aMax	:	TcVnVector4_DINT;	(* Returns the requested element *)
	END_VAR
	VAR_INPUT
		hrPrev	:	HRESULT;	(* HRESULT indicating the result of previous operations (If SUCCEEDED(hrPrev) equals false, no operation is executed.) *)
	END_VAR

END_FUNCTION

// Functions/Container Statistics/F_VN_MaxElementElementwise/F_VN_MaxElementElementwise_TcVnVector4_INT

	{attribute 'TcIecLibraryType'}
	{attribute 'external_name' := 'F_VN_MaxElementElementwise_TcVnVector4_INT_GUID_80CB51C0_655A_4390_F5B3_A79390A81269'}
	(* Gets the element wise maximum container element. *)
	FUNCTION F_VN_MaxElementElementwise_TcVnVector4_INT : HRESULT
	VAR_INPUT
		ipContainer	:	ITcVnContainer;	(* Source container *)
	END_VAR
	VAR_IN_OUT
		aMax	:	TcVnVector4_INT;	(* Returns the requested element *)
	END_VAR
	VAR_INPUT
		hrPrev	:	HRESULT;	(* HRESULT indicating the result of previous operations (If SUCCEEDED(hrPrev) equals false, no operation is executed.) *)
	END_VAR

END_FUNCTION

// Functions/Container Statistics/F_VN_MaxElementElementwise/F_VN_MaxElementElementwise_TcVnVector4_LREAL

	{attribute 'TcIecLibraryType'}
	{attribute 'external_name' := 'F_VN_MaxElementElementwise_TcVnVector4_LREAL_GUID_68EB68AC_BC03_4E8E_FDAA_B0FE14AD2C3D'}
	(* Gets the element wise maximum container element. *)
	FUNCTION F_VN_MaxElementElementwise_TcVnVector4_LREAL : HRESULT
	VAR_INPUT
		ipContainer	:	ITcVnContainer;	(* Source container *)
	END_VAR
	VAR_IN_OUT
		aMax	:	TcVnVector4_LREAL;	(* Returns the requested element *)
	END_VAR
	VAR_INPUT
		hrPrev	:	HRESULT;	(* HRESULT indicating the result of previous operations (If SUCCEEDED(hrPrev) equals false, no operation is executed.) *)
	END_VAR

END_FUNCTION

// Functions/Container Statistics/F_VN_MaxElementElementwise/F_VN_MaxElementElementwise_TcVnVector4_SINT

	{attribute 'TcIecLibraryType'}
	{attribute 'external_name' := 'F_VN_MaxElementElementwise_TcVnVector4_SINT_GUID_245A952C_302C_4494_EAF8_1A974CDD6018'}
	(* Gets the element wise maximum container element. *)
	FUNCTION F_VN_MaxElementElementwise_TcVnVector4_SINT : HRESULT
	VAR_INPUT
		ipContainer	:	ITcVnContainer;	(* Source container *)
	END_VAR
	VAR_IN_OUT
		aMax	:	TcVnVector4_SINT;	(* Returns the requested element *)
	END_VAR
	VAR_INPUT
		hrPrev	:	HRESULT;	(* HRESULT indicating the result of previous operations (If SUCCEEDED(hrPrev) equals false, no operation is executed.) *)
	END_VAR

END_FUNCTION

// Functions/Container Statistics/F_VN_MaxElementElementwise/F_VN_MaxElementElementwise_TcVnVector4_UINT

	{attribute 'TcIecLibraryType'}
	{attribute 'external_name' := 'F_VN_MaxElementElementwise_TcVnVector4_UINT_GUID_FA006A5C_1BC7_491A_F54F_D492797A56D3'}
	(* Gets the element wise maximum container element. *)
	FUNCTION F_VN_MaxElementElementwise_TcVnVector4_UINT : HRESULT
	VAR_INPUT
		ipContainer	:	ITcVnContainer;	(* Source container *)
	END_VAR
	VAR_IN_OUT
		aMax	:	TcVnVector4_UINT;	(* Returns the requested element *)
	END_VAR
	VAR_INPUT
		hrPrev	:	HRESULT;	(* HRESULT indicating the result of previous operations (If SUCCEEDED(hrPrev) equals false, no operation is executed.) *)
	END_VAR

END_FUNCTION

// Functions/Container Statistics/F_VN_MaxElementElementwise/F_VN_MaxElementElementwise_TcVnVector4_USINT

	{attribute 'TcIecLibraryType'}
	{attribute 'external_name' := 'F_VN_MaxElementElementwise_TcVnVector4_USINT_GUID_03D9B166_C005_43E8_D46E_D405E57F63CC'}
	(* Gets the element wise maximum container element. *)
	FUNCTION F_VN_MaxElementElementwise_TcVnVector4_USINT : HRESULT
	VAR_INPUT
		ipContainer	:	ITcVnContainer;	(* Source container *)
	END_VAR
	VAR_IN_OUT
		aMax	:	TcVnVector4_USINT;	(* Returns the requested element *)
	END_VAR
	VAR_INPUT
		hrPrev	:	HRESULT;	(* HRESULT indicating the result of previous operations (If SUCCEEDED(hrPrev) equals false, no operation is executed.) *)
	END_VAR

END_FUNCTION

// Functions/Container Statistics/F_VN_MaxElementElementwise/F_VN_MaxElementElementwise_UDINT

	{attribute 'TcIecLibraryType'}
	{attribute 'external_name' := 'F_VN_MaxElementElementwise_UDINT_GUID_B0A69D66_FBA0_4A5B_E623_B903EF52870B'}
	(* Gets the element wise maximum container element. *)
	FUNCTION F_VN_MaxElementElementwise_UDINT : HRESULT
	VAR_INPUT
		ipContainer	:	ITcVnContainer;	(* Source container *)
	END_VAR
	VAR_IN_OUT
		nMax	:	UDINT;	(* Returns the requested element *)
	END_VAR
	VAR_INPUT
		hrPrev	:	HRESULT;	(* HRESULT indicating the result of previous operations (If SUCCEEDED(hrPrev) equals false, no operation is executed.) *)
	END_VAR

END_FUNCTION

// Functions/Container Statistics/F_VN_MaxElementElementwise/F_VN_MaxElementElementwise_UINT

	{attribute 'TcIecLibraryType'}
	{attribute 'external_name' := 'F_VN_MaxElementElementwise_UINT_GUID_B36815F9_D62F_49CD_C06A_412B9C703BD0'}
	(* Gets the element wise maximum container element. *)
	FUNCTION F_VN_MaxElementElementwise_UINT : HRESULT
	VAR_INPUT
		ipContainer	:	ITcVnContainer;	(* Source container *)
	END_VAR
	VAR_IN_OUT
		nMax	:	UINT;	(* Returns the requested element *)
	END_VAR
	VAR_INPUT
		hrPrev	:	HRESULT;	(* HRESULT indicating the result of previous operations (If SUCCEEDED(hrPrev) equals false, no operation is executed.) *)
	END_VAR

END_FUNCTION

// Functions/Container Statistics/F_VN_MaxElementElementwise/F_VN_MaxElementElementwise_ULINT

	{attribute 'TcIecLibraryType'}
	{attribute 'external_name' := 'F_VN_MaxElementElementwise_ULINT_GUID_E6BA466A_541B_4E95_EC74_E01888F0967D'}
	(* Gets the element wise maximum container element. *)
	FUNCTION F_VN_MaxElementElementwise_ULINT : HRESULT
	VAR_INPUT
		ipContainer	:	ITcVnContainer;	(* Source container *)
	END_VAR
	VAR_IN_OUT
		nMax	:	ULINT;	(* Returns the requested element *)
	END_VAR
	VAR_INPUT
		hrPrev	:	HRESULT;	(* HRESULT indicating the result of previous operations (If SUCCEEDED(hrPrev) equals false, no operation is executed.) *)
	END_VAR

END_FUNCTION

// Functions/Container Statistics/F_VN_MaxElementElementwise/F_VN_MaxElementElementwise_USINT

	{attribute 'TcIecLibraryType'}
	{attribute 'external_name' := 'F_VN_MaxElementElementwise_USINT_GUID_FA08EB1B_7358_4A77_FC22_C56FC4D13D49'}
	(* Gets the element wise maximum container element. *)
	FUNCTION F_VN_MaxElementElementwise_USINT : HRESULT
	VAR_INPUT
		ipContainer	:	ITcVnContainer;	(* Source container *)
	END_VAR
	VAR_IN_OUT
		nMax	:	USINT;	(* Returns the requested element *)
	END_VAR
	VAR_INPUT
		hrPrev	:	HRESULT;	(* HRESULT indicating the result of previous operations (If SUCCEEDED(hrPrev) equals false, no operation is executed.) *)
	END_VAR

END_FUNCTION

// Functions/Container Statistics/F_VN_MedianElementElementwise/F_VN_MedianElementElementwise_DINT

	{attribute 'TcIecLibraryType'}
	{attribute 'external_name' := 'F_VN_MedianElementElementwise_DINT_GUID_B6479066_DD04_48F4_F717_9E8A090BE208'}
	(* Gets the element wise median container element. *)
	FUNCTION F_VN_MedianElementElementwise_DINT : HRESULT
	VAR_INPUT
		ipContainer	:	ITcVnContainer;	(* Source container *)
	END_VAR
	VAR_IN_OUT
		nMedian	:	DINT;	(* Returns the requested element *)
	END_VAR
	VAR_INPUT
		hrPrev	:	HRESULT;	(* HRESULT indicating the result of previous operations (If SUCCEEDED(hrPrev) equals false, no operation is executed.) *)
	END_VAR

END_FUNCTION

// Functions/Container Statistics/F_VN_MedianElementElementwise/F_VN_MedianElementElementwise_INT

	{attribute 'TcIecLibraryType'}
	{attribute 'external_name' := 'F_VN_MedianElementElementwise_INT_GUID_54E7D16E_DAA5_4DFF_FB3D_3249D3BAA279'}
	(* Gets the element wise median container element. *)
	FUNCTION F_VN_MedianElementElementwise_INT : HRESULT
	VAR_INPUT
		ipContainer	:	ITcVnContainer;	(* Source container *)
	END_VAR
	VAR_IN_OUT
		nMedian	:	INT;	(* Returns the requested element *)
	END_VAR
	VAR_INPUT
		hrPrev	:	HRESULT;	(* HRESULT indicating the result of previous operations (If SUCCEEDED(hrPrev) equals false, no operation is executed.) *)
	END_VAR

END_FUNCTION

// Functions/Container Statistics/F_VN_MedianElementElementwise/F_VN_MedianElementElementwise_LREAL

	{attribute 'TcIecLibraryType'}
	{attribute 'external_name' := 'F_VN_MedianElementElementwise_LREAL_GUID_2A8C0845_A2AC_4341_D47F_55552E95EFF4'}
	(* Gets the element wise median container element. *)
	FUNCTION F_VN_MedianElementElementwise_LREAL : HRESULT
	VAR_INPUT
		ipContainer	:	ITcVnContainer;	(* Source container *)
	END_VAR
	VAR_IN_OUT
		fMedian	:	LREAL;	(* Returns the requested element *)
	END_VAR
	VAR_INPUT
		hrPrev	:	HRESULT;	(* HRESULT indicating the result of previous operations (If SUCCEEDED(hrPrev) equals false, no operation is executed.) *)
	END_VAR

END_FUNCTION

// Functions/Container Statistics/F_VN_MedianElementElementwise/F_VN_MedianElementElementwise_REAL

	{attribute 'TcIecLibraryType'}
	{attribute 'external_name' := 'F_VN_MedianElementElementwise_REAL_GUID_BE33EFFD_A6AD_4337_F353_C38D140704BC'}
	(* Gets the element wise median container element. *)
	FUNCTION F_VN_MedianElementElementwise_REAL : HRESULT
	VAR_INPUT
		ipContainer	:	ITcVnContainer;	(* Source container *)
	END_VAR
	VAR_IN_OUT
		fMedian	:	REAL;	(* Returns the requested element *)
	END_VAR
	VAR_INPUT
		hrPrev	:	HRESULT;	(* HRESULT indicating the result of previous operations (If SUCCEEDED(hrPrev) equals false, no operation is executed.) *)
	END_VAR

END_FUNCTION

// Functions/Container Statistics/F_VN_MedianElementElementwise/F_VN_MedianElementElementwise_SINT

	{attribute 'TcIecLibraryType'}
	{attribute 'external_name' := 'F_VN_MedianElementElementwise_SINT_GUID_3886489C_3CEE_47B5_DE9F_37BDED3FF052'}
	(* Gets the element wise median container element. *)
	FUNCTION F_VN_MedianElementElementwise_SINT : HRESULT
	VAR_INPUT
		ipContainer	:	ITcVnContainer;	(* Source container *)
	END_VAR
	VAR_IN_OUT
		nMedian	:	SINT;	(* Returns the requested element *)
	END_VAR
	VAR_INPUT
		hrPrev	:	HRESULT;	(* HRESULT indicating the result of previous operations (If SUCCEEDED(hrPrev) equals false, no operation is executed.) *)
	END_VAR

END_FUNCTION

// Functions/Container Statistics/F_VN_MedianElementElementwise/F_VN_MedianElementElementwise_TcVnPoint2_DINT

	{attribute 'TcIecLibraryType'}
	{attribute 'external_name' := 'F_VN_MedianElementElementwise_TcVnPoint2_DINT_GUID_3CB43A97_7C23_487E_FB7F_27B5DBC57F3F'}
	(* Gets the element wise median container element. *)
	FUNCTION F_VN_MedianElementElementwise_TcVnPoint2_DINT : HRESULT
	VAR_INPUT
		ipContainer	:	ITcVnContainer;	(* Source container *)
	END_VAR
	VAR_IN_OUT
		aMedian	:	TcVnPoint2_DINT;	(* Returns the requested element *)
	END_VAR
	VAR_INPUT
		hrPrev	:	HRESULT;	(* HRESULT indicating the result of previous operations (If SUCCEEDED(hrPrev) equals false, no operation is executed.) *)
	END_VAR

END_FUNCTION

// Functions/Container Statistics/F_VN_MedianElementElementwise/F_VN_MedianElementElementwise_TcVnPoint2_LREAL

	{attribute 'TcIecLibraryType'}
	{attribute 'external_name' := 'F_VN_MedianElementElementwise_TcVnPoint2_LREAL_GUID_C747D101_6288_4FFB_E2DB_A25A7E4EF5ED'}
	(* Gets the element wise median container element. *)
	FUNCTION F_VN_MedianElementElementwise_TcVnPoint2_LREAL : HRESULT
	VAR_INPUT
		ipContainer	:	ITcVnContainer;	(* Source container *)
	END_VAR
	VAR_IN_OUT
		aMedian	:	TcVnPoint2_LREAL;	(* Returns the requested element *)
	END_VAR
	VAR_INPUT
		hrPrev	:	HRESULT;	(* HRESULT indicating the result of previous operations (If SUCCEEDED(hrPrev) equals false, no operation is executed.) *)
	END_VAR

END_FUNCTION

// Functions/Container Statistics/F_VN_MedianElementElementwise/F_VN_MedianElementElementwise_TcVnPoint2_REAL

	{attribute 'TcIecLibraryType'}
	{attribute 'external_name' := 'F_VN_MedianElementElementwise_TcVnPoint2_REAL_GUID_67BE655C_1115_462E_D1EF_EBC4BAEC34ED'}
	(* Gets the element wise median container element. *)
	FUNCTION F_VN_MedianElementElementwise_TcVnPoint2_REAL : HRESULT
	VAR_INPUT
		ipContainer	:	ITcVnContainer;	(* Source container *)
	END_VAR
	VAR_IN_OUT
		aMedian	:	TcVnPoint2_REAL;	(* Returns the requested element *)
	END_VAR
	VAR_INPUT
		hrPrev	:	HRESULT;	(* HRESULT indicating the result of previous operations (If SUCCEEDED(hrPrev) equals false, no operation is executed.) *)
	END_VAR

END_FUNCTION

// Functions/Container Statistics/F_VN_MedianElementElementwise/F_VN_MedianElementElementwise_TcVnPoint3_LREAL

	{attribute 'TcIecLibraryType'}
	{attribute 'external_name' := 'F_VN_MedianElementElementwise_TcVnPoint3_LREAL_GUID_6EA72555_1A23_4895_E439_D7D00A8D3666'}
	(* Gets the element wise median container element. *)
	FUNCTION F_VN_MedianElementElementwise_TcVnPoint3_LREAL : HRESULT
	VAR_INPUT
		ipContainer	:	ITcVnContainer;	(* Source container *)
	END_VAR
	VAR_IN_OUT
		aMedian	:	TcVnPoint3_LREAL;	(* Returns the requested element *)
	END_VAR
	VAR_INPUT
		hrPrev	:	HRESULT;	(* HRESULT indicating the result of previous operations (If SUCCEEDED(hrPrev) equals false, no operation is executed.) *)
	END_VAR

END_FUNCTION

// Functions/Container Statistics/F_VN_MedianElementElementwise/F_VN_MedianElementElementwise_TcVnPoint3_REAL

	{attribute 'TcIecLibraryType'}
	{attribute 'external_name' := 'F_VN_MedianElementElementwise_TcVnPoint3_REAL_GUID_EA823E13_4FA9_4B06_EBA7_434DCA0A5495'}
	(* Gets the element wise median container element. *)
	FUNCTION F_VN_MedianElementElementwise_TcVnPoint3_REAL : HRESULT
	VAR_INPUT
		ipContainer	:	ITcVnContainer;	(* Source container *)
	END_VAR
	VAR_IN_OUT
		aMedian	:	TcVnPoint3_REAL;	(* Returns the requested element *)
	END_VAR
	VAR_INPUT
		hrPrev	:	HRESULT;	(* HRESULT indicating the result of previous operations (If SUCCEEDED(hrPrev) equals false, no operation is executed.) *)
	END_VAR

END_FUNCTION

// Functions/Container Statistics/F_VN_MedianElementElementwise/F_VN_MedianElementElementwise_TcVnVector2_DINT

	{attribute 'TcIecLibraryType'}
	{attribute 'external_name' := 'F_VN_MedianElementElementwise_TcVnVector2_DINT_GUID_11AA23CC_9F9A_4F5C_D623_AE0E682B1785'}
	(* Gets the element wise median container element. *)
	FUNCTION F_VN_MedianElementElementwise_TcVnVector2_DINT : HRESULT
	VAR_INPUT
		ipContainer	:	ITcVnContainer;	(* Source container *)
	END_VAR
	VAR_IN_OUT
		aMedian	:	TcVnVector2_DINT;	(* Returns the requested element *)
	END_VAR
	VAR_INPUT
		hrPrev	:	HRESULT;	(* HRESULT indicating the result of previous operations (If SUCCEEDED(hrPrev) equals false, no operation is executed.) *)
	END_VAR

END_FUNCTION

// Functions/Container Statistics/F_VN_MedianElementElementwise/F_VN_MedianElementElementwise_TcVnVector2_INT

	{attribute 'TcIecLibraryType'}
	{attribute 'external_name' := 'F_VN_MedianElementElementwise_TcVnVector2_INT_GUID_C4302285_8AC8_4E74_E908_855CB2E4D1A8'}
	(* Gets the element wise median container element. *)
	FUNCTION F_VN_MedianElementElementwise_TcVnVector2_INT : HRESULT
	VAR_INPUT
		ipContainer	:	ITcVnContainer;	(* Source container *)
	END_VAR
	VAR_IN_OUT
		aMedian	:	TcVnVector2_INT;	(* Returns the requested element *)
	END_VAR
	VAR_INPUT
		hrPrev	:	HRESULT;	(* HRESULT indicating the result of previous operations (If SUCCEEDED(hrPrev) equals false, no operation is executed.) *)
	END_VAR

END_FUNCTION

// Functions/Container Statistics/F_VN_MedianElementElementwise/F_VN_MedianElementElementwise_TcVnVector2_REAL

	{attribute 'TcIecLibraryType'}
	{attribute 'external_name' := 'F_VN_MedianElementElementwise_TcVnVector2_REAL_GUID_1904A974_DBAF_47D0_DE6B_6DA50DCFF127'}
	(* Gets the element wise median container element. *)
	FUNCTION F_VN_MedianElementElementwise_TcVnVector2_REAL : HRESULT
	VAR_INPUT
		ipContainer	:	ITcVnContainer;	(* Source container *)
	END_VAR
	VAR_IN_OUT
		aMedian	:	TcVnVector2_REAL;	(* Returns the requested element *)
	END_VAR
	VAR_INPUT
		hrPrev	:	HRESULT;	(* HRESULT indicating the result of previous operations (If SUCCEEDED(hrPrev) equals false, no operation is executed.) *)
	END_VAR

END_FUNCTION

// Functions/Container Statistics/F_VN_MedianElementElementwise/F_VN_MedianElementElementwise_TcVnVector2_SINT

	{attribute 'TcIecLibraryType'}
	{attribute 'external_name' := 'F_VN_MedianElementElementwise_TcVnVector2_SINT_GUID_60CA0FF1_9AED_4F0A_CD37_99588C2348BA'}
	(* Gets the element wise median container element. *)
	FUNCTION F_VN_MedianElementElementwise_TcVnVector2_SINT : HRESULT
	VAR_INPUT
		ipContainer	:	ITcVnContainer;	(* Source container *)
	END_VAR
	VAR_IN_OUT
		aMedian	:	TcVnVector2_SINT;	(* Returns the requested element *)
	END_VAR
	VAR_INPUT
		hrPrev	:	HRESULT;	(* HRESULT indicating the result of previous operations (If SUCCEEDED(hrPrev) equals false, no operation is executed.) *)
	END_VAR

END_FUNCTION

// Functions/Container Statistics/F_VN_MedianElementElementwise/F_VN_MedianElementElementwise_TcVnVector2_UINT

	{attribute 'TcIecLibraryType'}
	{attribute 'external_name' := 'F_VN_MedianElementElementwise_TcVnVector2_UINT_GUID_EFB56105_47D9_4CC4_E1E2_60E6E3763DEC'}
	(* Gets the element wise median container element. *)
	FUNCTION F_VN_MedianElementElementwise_TcVnVector2_UINT : HRESULT
	VAR_INPUT
		ipContainer	:	ITcVnContainer;	(* Source container *)
	END_VAR
	VAR_IN_OUT
		aMedian	:	TcVnVector2_UINT;	(* Returns the requested element *)
	END_VAR
	VAR_INPUT
		hrPrev	:	HRESULT;	(* HRESULT indicating the result of previous operations (If SUCCEEDED(hrPrev) equals false, no operation is executed.) *)
	END_VAR

END_FUNCTION

// Functions/Container Statistics/F_VN_MedianElementElementwise/F_VN_MedianElementElementwise_TcVnVector2_USINT

	{attribute 'TcIecLibraryType'}
	{attribute 'external_name' := 'F_VN_MedianElementElementwise_TcVnVector2_USINT_GUID_BA9D0C33_1D78_4CB2_D15A_67F4157D7FD8'}
	(* Gets the element wise median container element. *)
	FUNCTION F_VN_MedianElementElementwise_TcVnVector2_USINT : HRESULT
	VAR_INPUT
		ipContainer	:	ITcVnContainer;	(* Source container *)
	END_VAR
	VAR_IN_OUT
		aMedian	:	TcVnVector2_USINT;	(* Returns the requested element *)
	END_VAR
	VAR_INPUT
		hrPrev	:	HRESULT;	(* HRESULT indicating the result of previous operations (If SUCCEEDED(hrPrev) equals false, no operation is executed.) *)
	END_VAR

END_FUNCTION

// Functions/Container Statistics/F_VN_MedianElementElementwise/F_VN_MedianElementElementwise_TcVnVector3_INT

	{attribute 'TcIecLibraryType'}
	{attribute 'external_name' := 'F_VN_MedianElementElementwise_TcVnVector3_INT_GUID_D33BC0D5_C1C1_426C_E347_CCBAEB5D3840'}
	(* Gets the element wise median container element. *)
	FUNCTION F_VN_MedianElementElementwise_TcVnVector3_INT : HRESULT
	VAR_INPUT
		ipContainer	:	ITcVnContainer;	(* Source container *)
	END_VAR
	VAR_IN_OUT
		aMedian	:	TcVnVector3_INT;	(* Returns the requested element *)
	END_VAR
	VAR_INPUT
		hrPrev	:	HRESULT;	(* HRESULT indicating the result of previous operations (If SUCCEEDED(hrPrev) equals false, no operation is executed.) *)
	END_VAR

END_FUNCTION

// Functions/Container Statistics/F_VN_MedianElementElementwise/F_VN_MedianElementElementwise_TcVnVector3_REAL

	{attribute 'TcIecLibraryType'}
	{attribute 'external_name' := 'F_VN_MedianElementElementwise_TcVnVector3_REAL_GUID_D1745B3D_E1E1_4EA1_DB57_2A024E56C0C8'}
	(* Gets the element wise median container element. *)
	FUNCTION F_VN_MedianElementElementwise_TcVnVector3_REAL : HRESULT
	VAR_INPUT
		ipContainer	:	ITcVnContainer;	(* Source container *)
	END_VAR
	VAR_IN_OUT
		aMedian	:	TcVnVector3_REAL;	(* Returns the requested element *)
	END_VAR
	VAR_INPUT
		hrPrev	:	HRESULT;	(* HRESULT indicating the result of previous operations (If SUCCEEDED(hrPrev) equals false, no operation is executed.) *)
	END_VAR

END_FUNCTION

// Functions/Container Statistics/F_VN_MedianElementElementwise/F_VN_MedianElementElementwise_TcVnVector3_SINT

	{attribute 'TcIecLibraryType'}
	{attribute 'external_name' := 'F_VN_MedianElementElementwise_TcVnVector3_SINT_GUID_0EDAC3EB_377E_42B4_CD41_64DD92927E34'}
	(* Gets the element wise median container element. *)
	FUNCTION F_VN_MedianElementElementwise_TcVnVector3_SINT : HRESULT
	VAR_INPUT
		ipContainer	:	ITcVnContainer;	(* Source container *)
	END_VAR
	VAR_IN_OUT
		aMedian	:	TcVnVector3_SINT;	(* Returns the requested element *)
	END_VAR
	VAR_INPUT
		hrPrev	:	HRESULT;	(* HRESULT indicating the result of previous operations (If SUCCEEDED(hrPrev) equals false, no operation is executed.) *)
	END_VAR

END_FUNCTION

// Functions/Container Statistics/F_VN_MedianElementElementwise/F_VN_MedianElementElementwise_TcVnVector3_UINT

	{attribute 'TcIecLibraryType'}
	{attribute 'external_name' := 'F_VN_MedianElementElementwise_TcVnVector3_UINT_GUID_373299A6_7E7C_4807_DD76_D33AB50767E0'}
	(* Gets the element wise median container element. *)
	FUNCTION F_VN_MedianElementElementwise_TcVnVector3_UINT : HRESULT
	VAR_INPUT
		ipContainer	:	ITcVnContainer;	(* Source container *)
	END_VAR
	VAR_IN_OUT
		aMedian	:	TcVnVector3_UINT;	(* Returns the requested element *)
	END_VAR
	VAR_INPUT
		hrPrev	:	HRESULT;	(* HRESULT indicating the result of previous operations (If SUCCEEDED(hrPrev) equals false, no operation is executed.) *)
	END_VAR

END_FUNCTION

// Functions/Container Statistics/F_VN_MedianElementElementwise/F_VN_MedianElementElementwise_TcVnVector3_USINT

	{attribute 'TcIecLibraryType'}
	{attribute 'external_name' := 'F_VN_MedianElementElementwise_TcVnVector3_USINT_GUID_93628E02_3310_40E9_D230_28353A2A7B9A'}
	(* Gets the element wise median container element. *)
	FUNCTION F_VN_MedianElementElementwise_TcVnVector3_USINT : HRESULT
	VAR_INPUT
		ipContainer	:	ITcVnContainer;	(* Source container *)
	END_VAR
	VAR_IN_OUT
		aMedian	:	TcVnVector3_USINT;	(* Returns the requested element *)
	END_VAR
	VAR_INPUT
		hrPrev	:	HRESULT;	(* HRESULT indicating the result of previous operations (If SUCCEEDED(hrPrev) equals false, no operation is executed.) *)
	END_VAR

END_FUNCTION

// Functions/Container Statistics/F_VN_MedianElementElementwise/F_VN_MedianElementElementwise_TcVnVector4_DINT

	{attribute 'TcIecLibraryType'}
	{attribute 'external_name' := 'F_VN_MedianElementElementwise_TcVnVector4_DINT_GUID_F040BDF0_393F_45AF_D875_4AEEFBB3F8F4'}
	(* Gets the element wise median container element. *)
	FUNCTION F_VN_MedianElementElementwise_TcVnVector4_DINT : HRESULT
	VAR_INPUT
		ipContainer	:	ITcVnContainer;	(* Source container *)
	END_VAR
	VAR_IN_OUT
		aMedian	:	TcVnVector4_DINT;	(* Returns the requested element *)
	END_VAR
	VAR_INPUT
		hrPrev	:	HRESULT;	(* HRESULT indicating the result of previous operations (If SUCCEEDED(hrPrev) equals false, no operation is executed.) *)
	END_VAR

END_FUNCTION

// Functions/Container Statistics/F_VN_MedianElementElementwise/F_VN_MedianElementElementwise_TcVnVector4_INT

	{attribute 'TcIecLibraryType'}
	{attribute 'external_name' := 'F_VN_MedianElementElementwise_TcVnVector4_INT_GUID_CB96BB71_572C_4D94_CFEC_8464B92AF59C'}
	(* Gets the element wise median container element. *)
	FUNCTION F_VN_MedianElementElementwise_TcVnVector4_INT : HRESULT
	VAR_INPUT
		ipContainer	:	ITcVnContainer;	(* Source container *)
	END_VAR
	VAR_IN_OUT
		aMedian	:	TcVnVector4_INT;	(* Returns the requested element *)
	END_VAR
	VAR_INPUT
		hrPrev	:	HRESULT;	(* HRESULT indicating the result of previous operations (If SUCCEEDED(hrPrev) equals false, no operation is executed.) *)
	END_VAR

END_FUNCTION

// Functions/Container Statistics/F_VN_MedianElementElementwise/F_VN_MedianElementElementwise_TcVnVector4_LREAL

	{attribute 'TcIecLibraryType'}
	{attribute 'external_name' := 'F_VN_MedianElementElementwise_TcVnVector4_LREAL_GUID_FD8B141E_625C_4E20_E76F_C57C5EB11709'}
	(* Gets the element wise median container element. *)
	FUNCTION F_VN_MedianElementElementwise_TcVnVector4_LREAL : HRESULT
	VAR_INPUT
		ipContainer	:	ITcVnContainer;	(* Source container *)
	END_VAR
	VAR_IN_OUT
		aMedian	:	TcVnVector4_LREAL;	(* Returns the requested element *)
	END_VAR
	VAR_INPUT
		hrPrev	:	HRESULT;	(* HRESULT indicating the result of previous operations (If SUCCEEDED(hrPrev) equals false, no operation is executed.) *)
	END_VAR

END_FUNCTION

// Functions/Container Statistics/F_VN_MedianElementElementwise/F_VN_MedianElementElementwise_TcVnVector4_SINT

	{attribute 'TcIecLibraryType'}
	{attribute 'external_name' := 'F_VN_MedianElementElementwise_TcVnVector4_SINT_GUID_FE8445E2_29C2_4393_CFCF_4BCEB56226AB'}
	(* Gets the element wise median container element. *)
	FUNCTION F_VN_MedianElementElementwise_TcVnVector4_SINT : HRESULT
	VAR_INPUT
		ipContainer	:	ITcVnContainer;	(* Source container *)
	END_VAR
	VAR_IN_OUT
		aMedian	:	TcVnVector4_SINT;	(* Returns the requested element *)
	END_VAR
	VAR_INPUT
		hrPrev	:	HRESULT;	(* HRESULT indicating the result of previous operations (If SUCCEEDED(hrPrev) equals false, no operation is executed.) *)
	END_VAR

END_FUNCTION

// Functions/Container Statistics/F_VN_MedianElementElementwise/F_VN_MedianElementElementwise_TcVnVector4_UINT

	{attribute 'TcIecLibraryType'}
	{attribute 'external_name' := 'F_VN_MedianElementElementwise_TcVnVector4_UINT_GUID_9B50A5FB_4B50_43EA_DA71_F1D306756F26'}
	(* Gets the element wise median container element. *)
	FUNCTION F_VN_MedianElementElementwise_TcVnVector4_UINT : HRESULT
	VAR_INPUT
		ipContainer	:	ITcVnContainer;	(* Source container *)
	END_VAR
	VAR_IN_OUT
		aMedian	:	TcVnVector4_UINT;	(* Returns the requested element *)
	END_VAR
	VAR_INPUT
		hrPrev	:	HRESULT;	(* HRESULT indicating the result of previous operations (If SUCCEEDED(hrPrev) equals false, no operation is executed.) *)
	END_VAR

END_FUNCTION

// Functions/Container Statistics/F_VN_MedianElementElementwise/F_VN_MedianElementElementwise_TcVnVector4_USINT

	{attribute 'TcIecLibraryType'}
	{attribute 'external_name' := 'F_VN_MedianElementElementwise_TcVnVector4_USINT_GUID_59FF1399_779A_4D1F_E53F_CC343B919E4F'}
	(* Gets the element wise median container element. *)
	FUNCTION F_VN_MedianElementElementwise_TcVnVector4_USINT : HRESULT
	VAR_INPUT
		ipContainer	:	ITcVnContainer;	(* Source container *)
	END_VAR
	VAR_IN_OUT
		aMedian	:	TcVnVector4_USINT;	(* Returns the requested element *)
	END_VAR
	VAR_INPUT
		hrPrev	:	HRESULT;	(* HRESULT indicating the result of previous operations (If SUCCEEDED(hrPrev) equals false, no operation is executed.) *)
	END_VAR

END_FUNCTION

// Functions/Container Statistics/F_VN_MedianElementElementwise/F_VN_MedianElementElementwise_UDINT

	{attribute 'TcIecLibraryType'}
	{attribute 'external_name' := 'F_VN_MedianElementElementwise_UDINT_GUID_042AA97B_0973_47B6_DF14_02778655CF49'}
	(* Gets the element wise median container element. *)
	FUNCTION F_VN_MedianElementElementwise_UDINT : HRESULT
	VAR_INPUT
		ipContainer	:	ITcVnContainer;	(* Source container *)
	END_VAR
	VAR_IN_OUT
		nMedian	:	UDINT;	(* Returns the requested element *)
	END_VAR
	VAR_INPUT
		hrPrev	:	HRESULT;	(* HRESULT indicating the result of previous operations (If SUCCEEDED(hrPrev) equals false, no operation is executed.) *)
	END_VAR

END_FUNCTION

// Functions/Container Statistics/F_VN_MedianElementElementwise/F_VN_MedianElementElementwise_UINT

	{attribute 'TcIecLibraryType'}
	{attribute 'external_name' := 'F_VN_MedianElementElementwise_UINT_GUID_3593121F_1F8B_4176_C1C7_F777243AA8B7'}
	(* Gets the element wise median container element. *)
	FUNCTION F_VN_MedianElementElementwise_UINT : HRESULT
	VAR_INPUT
		ipContainer	:	ITcVnContainer;	(* Source container *)
	END_VAR
	VAR_IN_OUT
		nMedian	:	UINT;	(* Returns the requested element *)
	END_VAR
	VAR_INPUT
		hrPrev	:	HRESULT;	(* HRESULT indicating the result of previous operations (If SUCCEEDED(hrPrev) equals false, no operation is executed.) *)
	END_VAR

END_FUNCTION

// Functions/Container Statistics/F_VN_MedianElementElementwise/F_VN_MedianElementElementwise_ULINT

	{attribute 'TcIecLibraryType'}
	{attribute 'external_name' := 'F_VN_MedianElementElementwise_ULINT_GUID_1122A94C_3615_4A4E_E7E3_C0C4A0288629'}
	(* Gets the element wise median container element. *)
	FUNCTION F_VN_MedianElementElementwise_ULINT : HRESULT
	VAR_INPUT
		ipContainer	:	ITcVnContainer;	(* Source container *)
	END_VAR
	VAR_IN_OUT
		nMedian	:	ULINT;	(* Returns the requested element *)
	END_VAR
	VAR_INPUT
		hrPrev	:	HRESULT;	(* HRESULT indicating the result of previous operations (If SUCCEEDED(hrPrev) equals false, no operation is executed.) *)
	END_VAR

END_FUNCTION

// Functions/Container Statistics/F_VN_MedianElementElementwise/F_VN_MedianElementElementwise_USINT

	{attribute 'TcIecLibraryType'}
	{attribute 'external_name' := 'F_VN_MedianElementElementwise_USINT_GUID_B6799E66_B065_4865_F27F_63D278CB17AE'}
	(* Gets the element wise median container element. *)
	FUNCTION F_VN_MedianElementElementwise_USINT : HRESULT
	VAR_INPUT
		ipContainer	:	ITcVnContainer;	(* Source container *)
	END_VAR
	VAR_IN_OUT
		nMedian	:	USINT;	(* Returns the requested element *)
	END_VAR
	VAR_INPUT
		hrPrev	:	HRESULT;	(* HRESULT indicating the result of previous operations (If SUCCEEDED(hrPrev) equals false, no operation is executed.) *)
	END_VAR

END_FUNCTION

// Functions/Container Statistics/F_VN_MinElementElementwise/F_VN_MinElementElementwise_DINT

	{attribute 'TcIecLibraryType'}
	{attribute 'external_name' := 'F_VN_MinElementElementwise_DINT_GUID_E1BB67FE_A387_439A_CFAD_0E266E12ADE9'}
	(* Gets the element wise minimum container element. *)
	FUNCTION F_VN_MinElementElementwise_DINT : HRESULT
	VAR_INPUT
		ipContainer	:	ITcVnContainer;	(* Source container *)
	END_VAR
	VAR_IN_OUT
		nMin	:	DINT;	(* Returns the requested element *)
	END_VAR
	VAR_INPUT
		hrPrev	:	HRESULT;	(* HRESULT indicating the result of previous operations (If SUCCEEDED(hrPrev) equals false, no operation is executed.) *)
	END_VAR

END_FUNCTION

// Functions/Container Statistics/F_VN_MinElementElementwise/F_VN_MinElementElementwise_INT

	{attribute 'TcIecLibraryType'}
	{attribute 'external_name' := 'F_VN_MinElementElementwise_INT_GUID_94544767_5E9A_418A_FF39_63E053C47674'}
	(* Gets the element wise minimum container element. *)
	FUNCTION F_VN_MinElementElementwise_INT : HRESULT
	VAR_INPUT
		ipContainer	:	ITcVnContainer;	(* Source container *)
	END_VAR
	VAR_IN_OUT
		nMin	:	INT;	(* Returns the requested element *)
	END_VAR
	VAR_INPUT
		hrPrev	:	HRESULT;	(* HRESULT indicating the result of previous operations (If SUCCEEDED(hrPrev) equals false, no operation is executed.) *)
	END_VAR

END_FUNCTION

// Functions/Container Statistics/F_VN_MinElementElementwise/F_VN_MinElementElementwise_LREAL

	{attribute 'TcIecLibraryType'}
	{attribute 'external_name' := 'F_VN_MinElementElementwise_LREAL_GUID_5E389EE6_F8D3_4499_C7F0_E28A49DBAB47'}
	(* Gets the element wise minimum container element. *)
	FUNCTION F_VN_MinElementElementwise_LREAL : HRESULT
	VAR_INPUT
		ipContainer	:	ITcVnContainer;	(* Source container *)
	END_VAR
	VAR_IN_OUT
		fMin	:	LREAL;	(* Returns the requested element *)
	END_VAR
	VAR_INPUT
		hrPrev	:	HRESULT;	(* HRESULT indicating the result of previous operations (If SUCCEEDED(hrPrev) equals false, no operation is executed.) *)
	END_VAR

END_FUNCTION

// Functions/Container Statistics/F_VN_MinElementElementwise/F_VN_MinElementElementwise_REAL

	{attribute 'TcIecLibraryType'}
	{attribute 'external_name' := 'F_VN_MinElementElementwise_REAL_GUID_DAEB1347_85AE_4B08_F255_D660AE3E054B'}
	(* Gets the element wise minimum container element. *)
	FUNCTION F_VN_MinElementElementwise_REAL : HRESULT
	VAR_INPUT
		ipContainer	:	ITcVnContainer;	(* Source container *)
	END_VAR
	VAR_IN_OUT
		fMin	:	REAL;	(* Returns the requested element *)
	END_VAR
	VAR_INPUT
		hrPrev	:	HRESULT;	(* HRESULT indicating the result of previous operations (If SUCCEEDED(hrPrev) equals false, no operation is executed.) *)
	END_VAR

END_FUNCTION

// Functions/Container Statistics/F_VN_MinElementElementwise/F_VN_MinElementElementwise_SINT

	{attribute 'TcIecLibraryType'}
	{attribute 'external_name' := 'F_VN_MinElementElementwise_SINT_GUID_B1E0B48A_CDBF_4F51_C981_5EF6203BC4EC'}
	(* Gets the element wise minimum container element. *)
	FUNCTION F_VN_MinElementElementwise_SINT : HRESULT
	VAR_INPUT
		ipContainer	:	ITcVnContainer;	(* Source container *)
	END_VAR
	VAR_IN_OUT
		nMin	:	SINT;	(* Returns the requested element *)
	END_VAR
	VAR_INPUT
		hrPrev	:	HRESULT;	(* HRESULT indicating the result of previous operations (If SUCCEEDED(hrPrev) equals false, no operation is executed.) *)
	END_VAR

END_FUNCTION

// Functions/Container Statistics/F_VN_MinElementElementwise/F_VN_MinElementElementwise_TcVnPoint2_DINT

	{attribute 'TcIecLibraryType'}
	{attribute 'external_name' := 'F_VN_MinElementElementwise_TcVnPoint2_DINT_GUID_912458D4_350F_4ECB_CEC0_AF1A595526F6'}
	(* Gets the element wise minimum container element. *)
	FUNCTION F_VN_MinElementElementwise_TcVnPoint2_DINT : HRESULT
	VAR_INPUT
		ipContainer	:	ITcVnContainer;	(* Source container *)
	END_VAR
	VAR_IN_OUT
		aMin	:	TcVnPoint2_DINT;	(* Returns the requested element *)
	END_VAR
	VAR_INPUT
		hrPrev	:	HRESULT;	(* HRESULT indicating the result of previous operations (If SUCCEEDED(hrPrev) equals false, no operation is executed.) *)
	END_VAR

END_FUNCTION

// Functions/Container Statistics/F_VN_MinElementElementwise/F_VN_MinElementElementwise_TcVnPoint2_LREAL

	{attribute 'TcIecLibraryType'}
	{attribute 'external_name' := 'F_VN_MinElementElementwise_TcVnPoint2_LREAL_GUID_05117A73_701E_486C_F029_B0023ACE0736'}
	(* Gets the element wise minimum container element. *)
	FUNCTION F_VN_MinElementElementwise_TcVnPoint2_LREAL : HRESULT
	VAR_INPUT
		ipContainer	:	ITcVnContainer;	(* Source container *)
	END_VAR
	VAR_IN_OUT
		aMin	:	TcVnPoint2_LREAL;	(* Returns the requested element *)
	END_VAR
	VAR_INPUT
		hrPrev	:	HRESULT;	(* HRESULT indicating the result of previous operations (If SUCCEEDED(hrPrev) equals false, no operation is executed.) *)
	END_VAR

END_FUNCTION

// Functions/Container Statistics/F_VN_MinElementElementwise/F_VN_MinElementElementwise_TcVnPoint2_REAL

	{attribute 'TcIecLibraryType'}
	{attribute 'external_name' := 'F_VN_MinElementElementwise_TcVnPoint2_REAL_GUID_E52BAF66_2ECC_4F13_DE37_C923279E6893'}
	(* Gets the element wise minimum container element. *)
	FUNCTION F_VN_MinElementElementwise_TcVnPoint2_REAL : HRESULT
	VAR_INPUT
		ipContainer	:	ITcVnContainer;	(* Source container *)
	END_VAR
	VAR_IN_OUT
		aMin	:	TcVnPoint2_REAL;	(* Returns the requested element *)
	END_VAR
	VAR_INPUT
		hrPrev	:	HRESULT;	(* HRESULT indicating the result of previous operations (If SUCCEEDED(hrPrev) equals false, no operation is executed.) *)
	END_VAR

END_FUNCTION

// Functions/Container Statistics/F_VN_MinElementElementwise/F_VN_MinElementElementwise_TcVnPoint3_LREAL

	{attribute 'TcIecLibraryType'}
	{attribute 'external_name' := 'F_VN_MinElementElementwise_TcVnPoint3_LREAL_GUID_2FC6D558_98E9_477B_C78E_E7CC1ACCB159'}
	(* Gets the element wise minimum container element. *)
	FUNCTION F_VN_MinElementElementwise_TcVnPoint3_LREAL : HRESULT
	VAR_INPUT
		ipContainer	:	ITcVnContainer;	(* Source container *)
	END_VAR
	VAR_IN_OUT
		aMin	:	TcVnPoint3_LREAL;	(* Returns the requested element *)
	END_VAR
	VAR_INPUT
		hrPrev	:	HRESULT;	(* HRESULT indicating the result of previous operations (If SUCCEEDED(hrPrev) equals false, no operation is executed.) *)
	END_VAR

END_FUNCTION

// Functions/Container Statistics/F_VN_MinElementElementwise/F_VN_MinElementElementwise_TcVnPoint3_REAL

	{attribute 'TcIecLibraryType'}
	{attribute 'external_name' := 'F_VN_MinElementElementwise_TcVnPoint3_REAL_GUID_89839421_C380_49BB_F7CB_7385A9E5EBB6'}
	(* Gets the element wise minimum container element. *)
	FUNCTION F_VN_MinElementElementwise_TcVnPoint3_REAL : HRESULT
	VAR_INPUT
		ipContainer	:	ITcVnContainer;	(* Source container *)
	END_VAR
	VAR_IN_OUT
		aMin	:	TcVnPoint3_REAL;	(* Returns the requested element *)
	END_VAR
	VAR_INPUT
		hrPrev	:	HRESULT;	(* HRESULT indicating the result of previous operations (If SUCCEEDED(hrPrev) equals false, no operation is executed.) *)
	END_VAR

END_FUNCTION

// Functions/Container Statistics/F_VN_MinElementElementwise/F_VN_MinElementElementwise_TcVnVector2_DINT

	{attribute 'TcIecLibraryType'}
	{attribute 'external_name' := 'F_VN_MinElementElementwise_TcVnVector2_DINT_GUID_D51D3DE7_5A14_44B2_D419_60D79B52344F'}
	(* Gets the element wise minimum container element. *)
	FUNCTION F_VN_MinElementElementwise_TcVnVector2_DINT : HRESULT
	VAR_INPUT
		ipContainer	:	ITcVnContainer;	(* Source container *)
	END_VAR
	VAR_IN_OUT
		aMin	:	TcVnVector2_DINT;	(* Returns the requested element *)
	END_VAR
	VAR_INPUT
		hrPrev	:	HRESULT;	(* HRESULT indicating the result of previous operations (If SUCCEEDED(hrPrev) equals false, no operation is executed.) *)
	END_VAR

END_FUNCTION

// Functions/Container Statistics/F_VN_MinElementElementwise/F_VN_MinElementElementwise_TcVnVector2_INT

	{attribute 'TcIecLibraryType'}
	{attribute 'external_name' := 'F_VN_MinElementElementwise_TcVnVector2_INT_GUID_CE732325_9799_4495_D5B0_FE19A80F8538'}
	(* Gets the element wise minimum container element. *)
	FUNCTION F_VN_MinElementElementwise_TcVnVector2_INT : HRESULT
	VAR_INPUT
		ipContainer	:	ITcVnContainer;	(* Source container *)
	END_VAR
	VAR_IN_OUT
		aMin	:	TcVnVector2_INT;	(* Returns the requested element *)
	END_VAR
	VAR_INPUT
		hrPrev	:	HRESULT;	(* HRESULT indicating the result of previous operations (If SUCCEEDED(hrPrev) equals false, no operation is executed.) *)
	END_VAR

END_FUNCTION

// Functions/Container Statistics/F_VN_MinElementElementwise/F_VN_MinElementElementwise_TcVnVector2_REAL

	{attribute 'TcIecLibraryType'}
	{attribute 'external_name' := 'F_VN_MinElementElementwise_TcVnVector2_REAL_GUID_1AC17E86_B305_4E2D_CD95_880D61BB8B95'}
	(* Gets the element wise minimum container element. *)
	FUNCTION F_VN_MinElementElementwise_TcVnVector2_REAL : HRESULT
	VAR_INPUT
		ipContainer	:	ITcVnContainer;	(* Source container *)
	END_VAR
	VAR_IN_OUT
		aMin	:	TcVnVector2_REAL;	(* Returns the requested element *)
	END_VAR
	VAR_INPUT
		hrPrev	:	HRESULT;	(* HRESULT indicating the result of previous operations (If SUCCEEDED(hrPrev) equals false, no operation is executed.) *)
	END_VAR

END_FUNCTION

// Functions/Container Statistics/F_VN_MinElementElementwise/F_VN_MinElementElementwise_TcVnVector2_SINT

	{attribute 'TcIecLibraryType'}
	{attribute 'external_name' := 'F_VN_MinElementElementwise_TcVnVector2_SINT_GUID_DA202F6F_FEB9_4B59_FF83_6CD6DEF8271C'}
	(* Gets the element wise minimum container element. *)
	FUNCTION F_VN_MinElementElementwise_TcVnVector2_SINT : HRESULT
	VAR_INPUT
		ipContainer	:	ITcVnContainer;	(* Source container *)
	END_VAR
	VAR_IN_OUT
		aMin	:	TcVnVector2_SINT;	(* Returns the requested element *)
	END_VAR
	VAR_INPUT
		hrPrev	:	HRESULT;	(* HRESULT indicating the result of previous operations (If SUCCEEDED(hrPrev) equals false, no operation is executed.) *)
	END_VAR

END_FUNCTION

// Functions/Container Statistics/F_VN_MinElementElementwise/F_VN_MinElementElementwise_TcVnVector2_UINT

	{attribute 'TcIecLibraryType'}
	{attribute 'external_name' := 'F_VN_MinElementElementwise_TcVnVector2_UINT_GUID_1D30052B_84D6_4B9E_EAF3_3FA574165B52'}
	(* Gets the element wise minimum container element. *)
	FUNCTION F_VN_MinElementElementwise_TcVnVector2_UINT : HRESULT
	VAR_INPUT
		ipContainer	:	ITcVnContainer;	(* Source container *)
	END_VAR
	VAR_IN_OUT
		aMin	:	TcVnVector2_UINT;	(* Returns the requested element *)
	END_VAR
	VAR_INPUT
		hrPrev	:	HRESULT;	(* HRESULT indicating the result of previous operations (If SUCCEEDED(hrPrev) equals false, no operation is executed.) *)
	END_VAR

END_FUNCTION

// Functions/Container Statistics/F_VN_MinElementElementwise/F_VN_MinElementElementwise_TcVnVector2_USINT

	{attribute 'TcIecLibraryType'}
	{attribute 'external_name' := 'F_VN_MinElementElementwise_TcVnVector2_USINT_GUID_4B29469D_BA43_48C2_E4F7_7E6A1AED978C'}
	(* Gets the element wise minimum container element. *)
	FUNCTION F_VN_MinElementElementwise_TcVnVector2_USINT : HRESULT
	VAR_INPUT
		ipContainer	:	ITcVnContainer;	(* Source container *)
	END_VAR
	VAR_IN_OUT
		aMin	:	TcVnVector2_USINT;	(* Returns the requested element *)
	END_VAR
	VAR_INPUT
		hrPrev	:	HRESULT;	(* HRESULT indicating the result of previous operations (If SUCCEEDED(hrPrev) equals false, no operation is executed.) *)
	END_VAR

END_FUNCTION

// Functions/Container Statistics/F_VN_MinElementElementwise/F_VN_MinElementElementwise_TcVnVector3_INT

	{attribute 'TcIecLibraryType'}
	{attribute 'external_name' := 'F_VN_MinElementElementwise_TcVnVector3_INT_GUID_9FD22FB1_4AF6_424F_F420_F6C7ED5F1607'}
	(* Gets the element wise minimum container element. *)
	FUNCTION F_VN_MinElementElementwise_TcVnVector3_INT : HRESULT
	VAR_INPUT
		ipContainer	:	ITcVnContainer;	(* Source container *)
	END_VAR
	VAR_IN_OUT
		aMin	:	TcVnVector3_INT;	(* Returns the requested element *)
	END_VAR
	VAR_INPUT
		hrPrev	:	HRESULT;	(* HRESULT indicating the result of previous operations (If SUCCEEDED(hrPrev) equals false, no operation is executed.) *)
	END_VAR

END_FUNCTION

// Functions/Container Statistics/F_VN_MinElementElementwise/F_VN_MinElementElementwise_TcVnVector3_REAL

	{attribute 'TcIecLibraryType'}
	{attribute 'external_name' := 'F_VN_MinElementElementwise_TcVnVector3_REAL_GUID_5311AEC2_246E_4A6F_D17C_5BE92E8832E0'}
	(* Gets the element wise minimum container element. *)
	FUNCTION F_VN_MinElementElementwise_TcVnVector3_REAL : HRESULT
	VAR_INPUT
		ipContainer	:	ITcVnContainer;	(* Source container *)
	END_VAR
	VAR_IN_OUT
		aMin	:	TcVnVector3_REAL;	(* Returns the requested element *)
	END_VAR
	VAR_INPUT
		hrPrev	:	HRESULT;	(* HRESULT indicating the result of previous operations (If SUCCEEDED(hrPrev) equals false, no operation is executed.) *)
	END_VAR

END_FUNCTION

// Functions/Container Statistics/F_VN_MinElementElementwise/F_VN_MinElementElementwise_TcVnVector3_SINT

	{attribute 'TcIecLibraryType'}
	{attribute 'external_name' := 'F_VN_MinElementElementwise_TcVnVector3_SINT_GUID_FF568C65_7668_46FF_EB14_ED89F02FFE5B'}
	(* Gets the element wise minimum container element. *)
	FUNCTION F_VN_MinElementElementwise_TcVnVector3_SINT : HRESULT
	VAR_INPUT
		ipContainer	:	ITcVnContainer;	(* Source container *)
	END_VAR
	VAR_IN_OUT
		aMin	:	TcVnVector3_SINT;	(* Returns the requested element *)
	END_VAR
	VAR_INPUT
		hrPrev	:	HRESULT;	(* HRESULT indicating the result of previous operations (If SUCCEEDED(hrPrev) equals false, no operation is executed.) *)
	END_VAR

END_FUNCTION

// Functions/Container Statistics/F_VN_MinElementElementwise/F_VN_MinElementElementwise_TcVnVector3_UINT

	{attribute 'TcIecLibraryType'}
	{attribute 'external_name' := 'F_VN_MinElementElementwise_TcVnVector3_UINT_GUID_AD468625_B2A5_4CE2_F321_A8E8B25253F4'}
	(* Gets the element wise minimum container element. *)
	FUNCTION F_VN_MinElementElementwise_TcVnVector3_UINT : HRESULT
	VAR_INPUT
		ipContainer	:	ITcVnContainer;	(* Source container *)
	END_VAR
	VAR_IN_OUT
		aMin	:	TcVnVector3_UINT;	(* Returns the requested element *)
	END_VAR
	VAR_INPUT
		hrPrev	:	HRESULT;	(* HRESULT indicating the result of previous operations (If SUCCEEDED(hrPrev) equals false, no operation is executed.) *)
	END_VAR

END_FUNCTION

// Functions/Container Statistics/F_VN_MinElementElementwise/F_VN_MinElementElementwise_TcVnVector3_USINT

	{attribute 'TcIecLibraryType'}
	{attribute 'external_name' := 'F_VN_MinElementElementwise_TcVnVector3_USINT_GUID_F30ACE67_A3D7_4123_F155_E51B80F7B567'}
	(* Gets the element wise minimum container element. *)
	FUNCTION F_VN_MinElementElementwise_TcVnVector3_USINT : HRESULT
	VAR_INPUT
		ipContainer	:	ITcVnContainer;	(* Source container *)
	END_VAR
	VAR_IN_OUT
		aMin	:	TcVnVector3_USINT;	(* Returns the requested element *)
	END_VAR
	VAR_INPUT
		hrPrev	:	HRESULT;	(* HRESULT indicating the result of previous operations (If SUCCEEDED(hrPrev) equals false, no operation is executed.) *)
	END_VAR

END_FUNCTION

// Functions/Container Statistics/F_VN_MinElementElementwise/F_VN_MinElementElementwise_TcVnVector4_DINT

	{attribute 'TcIecLibraryType'}
	{attribute 'external_name' := 'F_VN_MinElementElementwise_TcVnVector4_DINT_GUID_D5A22E29_52F0_4C46_DC35_D0DA75208BD2'}
	(* Gets the element wise minimum container element. *)
	FUNCTION F_VN_MinElementElementwise_TcVnVector4_DINT : HRESULT
	VAR_INPUT
		ipContainer	:	ITcVnContainer;	(* Source container *)
	END_VAR
	VAR_IN_OUT
		aMin	:	TcVnVector4_DINT;	(* Returns the requested element *)
	END_VAR
	VAR_INPUT
		hrPrev	:	HRESULT;	(* HRESULT indicating the result of previous operations (If SUCCEEDED(hrPrev) equals false, no operation is executed.) *)
	END_VAR

END_FUNCTION

// Functions/Container Statistics/F_VN_MinElementElementwise/F_VN_MinElementElementwise_TcVnVector4_INT

	{attribute 'TcIecLibraryType'}
	{attribute 'external_name' := 'F_VN_MinElementElementwise_TcVnVector4_INT_GUID_6B8733E4_DEF7_4CC9_D56D_3F07316092E1'}
	(* Gets the element wise minimum container element. *)
	FUNCTION F_VN_MinElementElementwise_TcVnVector4_INT : HRESULT
	VAR_INPUT
		ipContainer	:	ITcVnContainer;	(* Source container *)
	END_VAR
	VAR_IN_OUT
		aMin	:	TcVnVector4_INT;	(* Returns the requested element *)
	END_VAR
	VAR_INPUT
		hrPrev	:	HRESULT;	(* HRESULT indicating the result of previous operations (If SUCCEEDED(hrPrev) equals false, no operation is executed.) *)
	END_VAR

END_FUNCTION

// Functions/Container Statistics/F_VN_MinElementElementwise/F_VN_MinElementElementwise_TcVnVector4_LREAL

	{attribute 'TcIecLibraryType'}
	{attribute 'external_name' := 'F_VN_MinElementElementwise_TcVnVector4_LREAL_GUID_5369237A_5786_4B88_F7C0_A40ACC572785'}
	(* Gets the element wise minimum container element. *)
	FUNCTION F_VN_MinElementElementwise_TcVnVector4_LREAL : HRESULT
	VAR_INPUT
		ipContainer	:	ITcVnContainer;	(* Source container *)
	END_VAR
	VAR_IN_OUT
		aMin	:	TcVnVector4_LREAL;	(* Returns the requested element *)
	END_VAR
	VAR_INPUT
		hrPrev	:	HRESULT;	(* HRESULT indicating the result of previous operations (If SUCCEEDED(hrPrev) equals false, no operation is executed.) *)
	END_VAR

END_FUNCTION

// Functions/Container Statistics/F_VN_MinElementElementwise/F_VN_MinElementElementwise_TcVnVector4_SINT

	{attribute 'TcIecLibraryType'}
	{attribute 'external_name' := 'F_VN_MinElementElementwise_TcVnVector4_SINT_GUID_8CF272D9_0772_4728_D405_001B18F1B349'}
	(* Gets the element wise minimum container element. *)
	FUNCTION F_VN_MinElementElementwise_TcVnVector4_SINT : HRESULT
	VAR_INPUT
		ipContainer	:	ITcVnContainer;	(* Source container *)
	END_VAR
	VAR_IN_OUT
		aMin	:	TcVnVector4_SINT;	(* Returns the requested element *)
	END_VAR
	VAR_INPUT
		hrPrev	:	HRESULT;	(* HRESULT indicating the result of previous operations (If SUCCEEDED(hrPrev) equals false, no operation is executed.) *)
	END_VAR

END_FUNCTION

// Functions/Container Statistics/F_VN_MinElementElementwise/F_VN_MinElementElementwise_TcVnVector4_UINT

	{attribute 'TcIecLibraryType'}
	{attribute 'external_name' := 'F_VN_MinElementElementwise_TcVnVector4_UINT_GUID_43290FE0_3102_4465_E98D_1CF0BAF5A9D2'}
	(* Gets the element wise minimum container element. *)
	FUNCTION F_VN_MinElementElementwise_TcVnVector4_UINT : HRESULT
	VAR_INPUT
		ipContainer	:	ITcVnContainer;	(* Source container *)
	END_VAR
	VAR_IN_OUT
		aMin	:	TcVnVector4_UINT;	(* Returns the requested element *)
	END_VAR
	VAR_INPUT
		hrPrev	:	HRESULT;	(* HRESULT indicating the result of previous operations (If SUCCEEDED(hrPrev) equals false, no operation is executed.) *)
	END_VAR

END_FUNCTION

// Functions/Container Statistics/F_VN_MinElementElementwise/F_VN_MinElementElementwise_TcVnVector4_USINT

	{attribute 'TcIecLibraryType'}
	{attribute 'external_name' := 'F_VN_MinElementElementwise_TcVnVector4_USINT_GUID_E4332C28_43B1_4C76_C5B0_1B3E2EEF7807'}
	(* Gets the element wise minimum container element. *)
	FUNCTION F_VN_MinElementElementwise_TcVnVector4_USINT : HRESULT
	VAR_INPUT
		ipContainer	:	ITcVnContainer;	(* Source container *)
	END_VAR
	VAR_IN_OUT
		aMin	:	TcVnVector4_USINT;	(* Returns the requested element *)
	END_VAR
	VAR_INPUT
		hrPrev	:	HRESULT;	(* HRESULT indicating the result of previous operations (If SUCCEEDED(hrPrev) equals false, no operation is executed.) *)
	END_VAR

END_FUNCTION

// Functions/Container Statistics/F_VN_MinElementElementwise/F_VN_MinElementElementwise_UDINT

	{attribute 'TcIecLibraryType'}
	{attribute 'external_name' := 'F_VN_MinElementElementwise_UDINT_GUID_EF3B2A64_610D_4B39_F43E_24490A0C0F59'}
	(* Gets the element wise minimum container element. *)
	FUNCTION F_VN_MinElementElementwise_UDINT : HRESULT
	VAR_INPUT
		ipContainer	:	ITcVnContainer;	(* Source container *)
	END_VAR
	VAR_IN_OUT
		nMin	:	UDINT;	(* Returns the requested element *)
	END_VAR
	VAR_INPUT
		hrPrev	:	HRESULT;	(* HRESULT indicating the result of previous operations (If SUCCEEDED(hrPrev) equals false, no operation is executed.) *)
	END_VAR

END_FUNCTION

// Functions/Container Statistics/F_VN_MinElementElementwise/F_VN_MinElementElementwise_UINT

	{attribute 'TcIecLibraryType'}
	{attribute 'external_name' := 'F_VN_MinElementElementwise_UINT_GUID_EEFC77E2_629E_4176_C323_CF8C653DE849'}
	(* Gets the element wise minimum container element. *)
	FUNCTION F_VN_MinElementElementwise_UINT : HRESULT
	VAR_INPUT
		ipContainer	:	ITcVnContainer;	(* Source container *)
	END_VAR
	VAR_IN_OUT
		nMin	:	UINT;	(* Returns the requested element *)
	END_VAR
	VAR_INPUT
		hrPrev	:	HRESULT;	(* HRESULT indicating the result of previous operations (If SUCCEEDED(hrPrev) equals false, no operation is executed.) *)
	END_VAR

END_FUNCTION

// Functions/Container Statistics/F_VN_MinElementElementwise/F_VN_MinElementElementwise_ULINT

	{attribute 'TcIecLibraryType'}
	{attribute 'external_name' := 'F_VN_MinElementElementwise_ULINT_GUID_7FD25639_574C_458B_FCFA_DC3853CD5908'}
	(* Gets the element wise minimum container element. *)
	FUNCTION F_VN_MinElementElementwise_ULINT : HRESULT
	VAR_INPUT
		ipContainer	:	ITcVnContainer;	(* Source container *)
	END_VAR
	VAR_IN_OUT
		nMin	:	ULINT;	(* Returns the requested element *)
	END_VAR
	VAR_INPUT
		hrPrev	:	HRESULT;	(* HRESULT indicating the result of previous operations (If SUCCEEDED(hrPrev) equals false, no operation is executed.) *)
	END_VAR

END_FUNCTION

// Functions/Container Statistics/F_VN_MinElementElementwise/F_VN_MinElementElementwise_USINT

	{attribute 'TcIecLibraryType'}
	{attribute 'external_name' := 'F_VN_MinElementElementwise_USINT_GUID_AFDCDF3F_E3CC_49C5_C26C_E27F0C7D5F9E'}
	(* Gets the element wise minimum container element. *)
	FUNCTION F_VN_MinElementElementwise_USINT : HRESULT
	VAR_INPUT
		ipContainer	:	ITcVnContainer;	(* Source container *)
	END_VAR
	VAR_IN_OUT
		nMin	:	USINT;	(* Returns the requested element *)
	END_VAR
	VAR_INPUT
		hrPrev	:	HRESULT;	(* HRESULT indicating the result of previous operations (If SUCCEEDED(hrPrev) equals false, no operation is executed.) *)
	END_VAR

END_FUNCTION
